TYPE "FANUC_OUTPUTS"
// stored: IsFailsafeCompliant false
   STRUCT
      SYSTEM_SIGNAL : Struct
         SYS_CMD_ENABLE : Bool;   // MACHINE HEARTBEAT (MACHINE TO GANTRY) / COMMAND ENABLE
         SYS_READY : Bool;   // SYSTEM READY
         SYS_PRG_RUNNING : Bool;   // MACHINE EMERGENCY STOP OK (MACHINE TO GANTRY) / PROGRAM RUNNING
         SYS_PRG_PAUSED : Bool;   // MACHINE SAFETY GATES OK (LOCKED)(MACHINE TO GANTRY) / PROGRAM PAUSED
         SYS_MOTION_HELD : Bool;   // MACHINE IN MANUAL MODE (MACHINE TO GANTRY) / MOTION HELD
         SYS_FAULT : Bool;   // MACHINE IN AUTO MODE(MACHINE TO GANTRY) / FAULT
         SYS_TP_ENABLED : Bool;   // MACHINE AUTO CYCLE RUNNING (MACHINE TO GANTRY) / TP ENABLED
         SYS_HOLD : Bool;   // MACHINE IS IN WARMUP CYCLE (MACHINE TO GANTRY) / ROBOT HOLD
         SPARE_1_0 : Byte;   // MACHINE IN RUN OUT MODE (MACHINE TO GANTRY)
         SPARE_2_0 : Byte;   // MACHINE PART DEMAND SOON (MACHINE TO GANTRY)
         SPARE_3_0 : Byte;
      END_STRUCT;
      GENERAL_SIGNAL : Struct
         STYLE_INIT_ACK : Bool;   // GANTRY HEARTBEAT (GANTRY TO MACHINE) / ACKNOWLEDGE INITIATE STYLE
         IN_CYCLE : Bool;   // IN CYCLE
         REQ_TO_CONT : Bool;   // GANTRY EMERGENCY STOP OK (GANTRY TO MACHINE) / REQUEST TO CONTINUE
         DRY_CYCLE : Bool;   // DRY CYCLE MODE
         RBT_100_SPD : Bool;   // GANTRY IN MANUAL MODE (GANTRY TO MACHINE) / ROBOT 100% SPEED
         RBT_HEARTBEAT : Bool;   // GANTRY IN AUTO MODE (GANTRY TO MACHINE) / ROBOT HEARTBEAT SIGNAL
         "OP_PANEL_E-STOP" : Bool;   // GANTRY IN AUTO CYCLE RUNNING (GANTRY TO MACHINE) / OPERATOR PANEL E-STOP
         "TEACH_PENDANT_E-STOP" : Bool;   // GANTRY OVERHEAD DOOR CLOSED & LOCKED (GANTRY TO MACHINE) / TEACH PENDANT E-STOP
         EXT_ENABLED : Bool;   // GANTRY IN RUN OUT COMPLETE(GANTRY TO MACHINE) / EXTERNAL E-STOP
         DEAD_ENABLED : Bool;   // GANTRY CLEAR OF MACHINE (GANTRY TO MACHINE) / DEADMAN E-STOP
         "I/O_SIMULATE" : Bool;   // GANTRY CLEAR OF FIXTURE (GANTRY TO MACHINE) / I/O SIMULATED
         SRV_DISC_OFF : Bool;   // SERVO DISABLED OFF
         SRV_BATT_ALARM : Bool;   // LOW BATTERY ALARM ON SERVO
         TASK_OK : Bool;   // TASK OK
         STEP_MODE_ON : Bool;   // STEP MODE STATUS
         AUTO_MODE_ON : Bool;   // SELECTOR SWITCH IS SET TO AUTO
         T1_MODE_ON : Bool;   // SELECTOR SWITCH IS SET TO T1
         T2_MODE_ON : Bool;   // SELECTOR SWITCH IS SET TO T2
         FENCE_OPEN : Bool;   // FENCE IS OPEN
         INTERLOCK : Bool;   // ROBOT IN INTERLOCK
         ROUT_ACTIVE : Bool;   // ROUTER ACTIVE BIT
         FAULT_RSP_ACK : Bool;   // HMI OPTION FAULT RESPONSE
         DCS_SIGN_MATCH : Bool;   // DCS SIGNATURE MATCH
         REQ_DEC_CODE : Bool;   // REQUEST DECITION
         FLT_TASK_STOPPED : Bool;   // ROBOT TASK STOPPED
         FLT_COLLISION : Bool;   // ROBOT COLLITION FAULT
         FLT_BAD_PLC_INPUT : Bool;   // BAD PLC INPUT
         FLT_GRIP_LOW_PRS : Bool;   // ROBOT GRIPPER PRESSURE LOW
         FLT_BAD_OPTN : Bool;   // BAD PLC FAULT RESPONSE
         RECOV_AT_MAIN : Bool;   // RECOVERY POINTER TO MAIN
         FLT_USER_BIT_8 : Bool;   // USER DEFINABLE FAULT BIT
         SPARE_7_7 : Bool;
         SPARE_8_0 : Byte;
         SPARE_9_0 : Byte;
      END_STRUCT;
      PROGRAM : Struct
         STYLE_PROGRAM_ACK : Byte;   // GANTRY HEARTBEAT (GANTRY TO MACHINE) / SELECT STYLE PROGRAM ACKNOWLEDGE
         DEC_CODE_ACK : Byte;   // SELECT DECITION CODE ACKNOWLEDGE
         PART_TYPE_ACK : Byte;   // GANTRY EMERGENCY STOP OK (GANTRY TO MACHINE) / PART TYPE ACKNOWLEDGE
         SPARE_13_0 : Byte;   // GANTRY EMERGENCY STOP OK (GANTRY TO MACHINE)
      END_STRUCT;
      GRIPPERS : Struct
         T1_GRIPPER_A_OPEN_REQ : Bool;   // ROBOT TOOL 1 GRIPPER A OPEN REQUEST
         T1_GRIPPER_A_CLOSE_REQ : Bool;   // ROBOT TOOL 1 GRIPPER A CLOSE REQUEST
         SPARE_14_2 : Bool;
         SPARE_14_3 : Bool;
         T1_GRIPPER_A_OPEN : Bool;   // ROBOT TOOL 1 GRIPPER A OPEN
         T1_GRIPPER_A_CLOSED : Bool;   // ROBOT TOOL 1 GRIPPER A CLOSED
         SPARE_14_6 : Bool;
         SPARE_14_7 : Bool;
         T1_GRIPPER_B_OPEN_REQ : Bool;   // ROBOT TOOL 1 GRIPPER B OPEN REQUEST
         T1_GRIPPER_B_CLOSE_REQ : Bool;   // ROBOT TOOL 1 GRIPPER B CLOSE REQUEST
         SPARE_15_2 : Bool;
         SPARE_15_3 : Bool;
         T1_GRIPPER_B_OPEN : Bool;   // ROBOT TOOL 1 GRIPPER B OPEN
         T1_GRIPPER_B_CLOSED : Bool;   // ROBOT TOOL 1 GRIPPER B CLOSED
         SPARE_15_6 : Bool;
         SPARE_15_7 : Bool;
         T1_GRIPPER_C_OPEN_REQ : Bool;   // ROBOT TOOL 1 GRIPPER C OPEN REQUEST
         T1_GRIPPER_C_CLOSE_REQ : Bool;   // ROBOT TOOL 1 GRIPPER C CLOSE REQUEST
         SPARE_16_2 : Bool;
         SPARE_16_3 : Bool;
         T1_GRIPPER_C_OPEN : Bool;   // ROBOT TOOL 1 GRIPPER C OPEN
         T1_GRIPPER_C_CLOSED : Bool;   // ROBOT TOOL 1 GRIPPER C CLOSED
         SPARE_16_6 : Bool;
         SPARE_16_7 : Bool;
         T1_GRIPPER_D_OPEN_REQ : Bool;   // ROBOT TOOL 1 GRIPPER D OPEN REQUEST
         T1_GRIPPER_D_CLOSE_REQ : Bool;   // ROBOT TOOL 1 GRIPPER D CLOSE REQUEST
         SPARE_17_2 : Bool;
         SPARE_17_3 : Bool;
         T1_GRIPPER_D_OPEN : Bool;   // ROBOT TOOL 1 GRIPPER D OPEN
         T1_GRIPPER_D_CLOSED : Bool;   // ROBOT TOOL 1 GRIPPER D CLOSED
         SPARE_17_6 : Bool;
         SPARE_17_7 : Bool;
         T1_GRIPPER_E_OPEN_REQ : Bool;   // ROBOT TOOL 1 GRIPPER E OPEN REQUEST
         T1_GRIPPER_E_CLOSE_REQ : Bool;   // ROBOT TOOL 1 GRIPPER E CLOSE REQUEST
         SPARE_18_2 : Bool;
         SPARE_18_3 : Bool;
         T1_GRIPPER_E_OPEN : Bool;   // ROBOT TOOL 1 GRIPPER E OPEN
         T1_GRIPPER_E_CLOSED : Bool;   // ROBOT TOOL 1 GRIPPER E CLOSED
         SPARE_18_6 : Bool;
         SPARE_18_7 : Bool;
         T2_GRIPPER_A_OPEN_REQ : Bool;   // ROBOT TOOL 2 GRIPPER A OPEN REQUEST
         T2_GRIPPER_A_CLOSE_REQ : Bool;   // ROBOT TOOL 2 GRIPPER A CLOSE REQUEST
         SPARE_19_2 : Bool;
         SPARE_19_3 : Bool;
         T2_GRIPPER_A_OPEN : Bool;   // ROBOT TOOL 2 GRIPPER A OPEN
         T2_GRIPPER_A_CLOSED : Bool;   // ROBOT TOOL 2 GRIPPER A CLOSED
         SPARE_19_6 : Bool;
         SPARE_19_7 : Bool;
         T2_GRIPPER_B_OPEN_REQ : Bool;   // ROBOT TOOL 2 GRIPPER B OPEN REQUEST
         T2_GRIPPER_B_CLOSE_REQ : Bool;   // ROBOT TOOL 2 GRIPPER B CLOSE REQUEST
         SPARE_20_2 : Bool;
         SPARE_20_3 : Bool;
         T2_GRIPPER_B_OPEN : Bool;   // ROBOT TOOL 2 GRIPPER B OPEN
         T2_GRIPPER_B_CLOSED : Bool;   // ROBOT TOOL 2 GRIPPER B CLOSED
         SPARE_20_6 : Bool;
         SPARE_20_7 : Bool;
         T2_GRIPPER_C_OPEN_REQ : Bool;   // ROBOT TOOL 2 GRIPPER C OPEN REQUEST
         T2_GRIPPER_C_CLOSE_REQ : Bool;   // ROBOT TOOL 2 GRIPPER C CLOSE REQUEST
         SPARE_21_2 : Bool;
         SPARE_21_3 : Bool;
         T2_GRIPPER_C_OPEN : Bool;   // ROBOT TOOL 2 GRIPPER C OPEN
         T2_GRIPPER_C_CLOSED : Bool;   // ROBOT TOOL 2 GRIPPER C CLOSED
         SPARE_21_6 : Bool;
         SPARE_21_7 : Bool;
         T2_GRIPPER_D_OPEN_REQ : Bool;   // ROBOT TOOL 2 GRIPPER D OPEN REQUEST
         T2_GRIPPER_D_CLOSE_REQ : Bool;   // ROBOT TOOL 2 GRIPPER D CLOSE REQUEST
         SPARE_22_2 : Bool;
         SPARE_22_3 : Bool;
         T2_GRIPPER_D_OPEN : Bool;   // ROBOT TOOL 2 GRIPPER D OPEN
         T2_GRIPPER_D_CLOSED : Bool;   // ROBOT TOOL 2 GRIPPER D CLOSED
         SPARE_22_6 : Bool;
         SPARE_22_7 : Bool;
         T2_GRIPPER_E_OPEN_REQ : Bool;   // ROBOT TOOL 2 GRIPPER E OPEN REQUEST
         T2_GRIPPER_E_CLOSE_REQ : Bool;   // ROBOT TOOL 2 GRIPPER E CLOSE REQUEST
         SPARE_23_2 : Bool;
         SPARE_23_3 : Bool;
         T2_GRIPPER_E_OPEN : Bool;   // ROBOT TOOL 2 GRIPPER E OPEN
         T2_GRIPPER_E_CLOSED : Bool;   // ROBOT TOOL 2 GRIPPER E CLOSED
         SPARE_23_6 : Bool;
         SPARE_23_7 : Bool;
         T1_ALL_GRIPS_OPEN_REQ : Bool;   // ROBOT TOOL 1 OPEN ALL GRIPPERS REQUEST
         T1_ALL_GRIPS_CLOSE_REQ : Bool;   // ROBOT TOOL 1 CLOSE ALL GRIPPERS REQUEST
         T1_ALL_GRIPPERS_OPEN : Bool;   // ROBOT TOOL 1 ALL GRIPPERS OPEN
         T1_ALL_GRIPPERS_CLOSED : Bool;   // ROBOT TOOL 1 ALL GRIPPERS CLOSED
         SPARE_24_4 : Bool;
         SPARE_24_5 : Bool;
         SPARE_24_6 : Bool;
         SPARE_24_7 : Bool;
         T2_ALL_GRIPS_OPEN_REQ : Bool;   // ROBOT TOOL 2 CLOSE ALL GRIPPERS REQUEST
         T2_ALL_GRIPS_CLOSE_REQ : Bool;   // ROBOT TOOL 2 CLOSE ALL GRIPPERS REQUEST
         T2_ALL_GRIPPERS_OPEN : Bool;   // ROBOT TOOL 2 ALL GRIPPERS OPEN
         T2_ALL_GRIPPERS_CLOSED : Bool;   // ROBOT TOOL 2 ALL GRIPPERS CLOSED
         SPARE_25_4 : Bool;
         SPARE_25_5 : Bool;
         SPARE_25_6 : Bool;
         SPARE_25_7 : Bool;
         SPARE_26_0 : Byte;
         FAULT_NUMBER : Byte;   // FAULT RESPONSE
      END_STRUCT;
      CLEARS : Struct
         CLEAR_U_1_ACK : Bool;   // GANTRY HEARTBEAT (GANTRY TO MACHINE) / ROBOT OUT OF UNIT 1
         CLEAR_U_2_ACK : Bool;   // ROBOT OUT OF UNIT 2
         CLEAR_U_3_ACK : Bool;   // GANTRY EMERGENCY STOP OK (GANTRY TO MACHINE) / ROBOT OUT OF UNIT 3
         CLEAR_U_4_ACK : Bool;   // ROBOT OUT OF UNIT 4
         CLEAR_U_5_ACK : Bool;   // GANTRY IN MANUAL MODE (GANTRY TO MACHINE) / ROBOT OUT OF UNIT 5
         CLEAR_U_6_ACK : Bool;   // GANTRY IN AUTO MODE (GANTRY TO MACHINE) / ROBOT OUT OF UNIT 6
         CLEAR_U_7_ACK : Bool;   // GANTRY IN AUTO CYCLE RUNNING (GANTRY TO MACHINE) / ROBOT OUT OF UNIT 7
         CLEAR_U_8_ACK : Bool;   // GANTRY OVERHEAD DOOR CLOSED & LOCKED (GANTRY TO MACHINE) / ROBOT OUT OF UNIT 8
         CLEAR_U_9_ACK : Bool;   // GANTRY IN RUN OUT COMPLETE(GANTRY TO MACHINE) / ROBOT OUT OF UNIT 9
         CLEAR_U_10_ACK : Bool;   // GANTRY CLEAR OF MACHINE (GANTRY TO MACHINE) / ROBOT OUT OF UNIT 10
         SPARE_29_2 : Bool;   // GANTRY CLEAR OF FIXTURE (GANTRY TO MACHINE)
         SPARE_29_3 : Bool;
         SPARE_29_4 : Bool;
         SPARE_29_5 : Bool;   // GANTRY PART TYPE CHANGE REQUESTED (GANTRY TO MACHINE)
         SPARE_29_6 : Bool;   // GANTRY REQUEST MACHINE TO RUN WITH LOADED PARTS (GANTRY TO MACHINE)
         SPARE_29_7 : Bool;   // GANTRY RUN OUT REQUESTED (GANTRY TO MACHINE)
         SPARE_30_0 : Byte;
         SPARE_31_0 : Byte;
      END_STRUCT;
      TASKS : Struct
         TSK_COMPLETED_1 : Bool;   // GANTRY HEARTBEAT (GANTRY TO MACHINE) / ROBOT TASK 1 COMPLETED
         TSK_COMPLETED_2 : Bool;   // ROBOT TASK 2 COMPLETED
         TSK_COMPLETED_3 : Bool;   // GANTRY EMERGENCY STOP OK (GANTRY TO MACHINE) / ROBOT TASK 3 COMPLETED
         TSK_COMPLETED_4 : Bool;   // ROBOT TASK 4 COMPLETED
         TSK_COMPLETED_5 : Bool;   // GANTRY IN MANUAL MODE (GANTRY TO MACHINE) / ROBOT TASK 5 COMPLETED
         TSK_COMPLETED_6 : Bool;   // GANTRY IN AUTO MODE (GANTRY TO MACHINE) / ROBOT TASK 6 COMPLETED
         TSK_COMPLETED_7 : Bool;   // GANTRY IN AUTO CYCLE RUNNING (GANTRY TO MACHINE) / ROBOT TASK 7 COMPLETED
         TSK_COMPLETED_8 : Bool;   // GANTRY OVERHEAD DOOR CLOSED & LOCKED (GANTRY TO MACHINE) / ROBOT TASK 8 COMPLETED
         SPARE_33_0 : Byte;   // GANTRY IN RUN OUT COMPLETE(GANTRY TO MACHINE) / ROBOT TASK 9 COMPLETED
         SPARE_34_0 : Byte;   // GANTRY CLEAR OF MACHINE (GANTRY TO MACHINE) / ROBOT TASK 10 COMPLETED
         SPARE_35_0 : Byte;   // GANTRY CLEAR OF FIXTURE (GANTRY TO MACHINE)
         SPARE_36_0 : Byte;
         SPARE_37_0 : Byte;
         SPARE_38_0 : Byte;
         SPARE_39_0 : Byte;
      END_STRUCT;
      POSITIONS : Struct
         HOME : Bool;   // GANTRY HEARTBEAT (GANTRY TO MACHINE) / ROBOT AT HOME POSITION
         MAINT : Bool;   // ROBOT AT MAINTENANCE POSITION
         REPAIR : Bool;   // GANTRY EMERGENCY STOP OK (GANTRY TO MACHINE) / ROBOT AT REPAIRED POSITION
         ALIGN : Bool;   // ROBOT AT ALIGNED POSITION
         SHIP : Bool;   // GANTRY IN MANUAL MODE (GANTRY TO MACHINE) / ROBOT AT SHIPPED POSITION
         SPARE_38_5 : Bool;   // GANTRY IN AUTO MODE (GANTRY TO MACHINE)
         SPARE_38_6 : Bool;   // GANTRY IN AUTO CYCLE RUNNING (GANTRY TO MACHINE)
         SPARE_38_7 : Bool;   // GANTRY OVERHEAD DOOR CLOSED & LOCKED (GANTRY TO MACHINE)
         UNIT_1 : Bool;   // GANTRY OVERHEAD DOOR CLOSED & LOCKED (GANTRY TO MACHINE) / ROBOT AT POUNCE POSITION UNIT 1
         UNIT_2 : Bool;   // GANTRY OVERHEAD DOOR CLOSED & LOCKED (GANTRY TO MACHINE) / ROBOT AT POUNCE POSITION UNIT 2
         UNIT_3 : Bool;   // GANTRY OVERHEAD DOOR CLOSED & LOCKED (GANTRY TO MACHINE) / ROBOT AT POUNCE POSITION UNIT 3
         UNIT_4 : Bool;   // GANTRY OVERHEAD DOOR CLOSED & LOCKED (GANTRY TO MACHINE) / ROBOT AT POUNCE POSITION UNIT 4
         UNIT_5 : Bool;   // GANTRY OVERHEAD DOOR CLOSED & LOCKED (GANTRY TO MACHINE) / ROBOT AT POUNCE POSITION UNIT 5
         UNIT_6 : Bool;   // GANTRY IN RUN OUT COMPLETE(GANTRY TO MACHINE) / ROBOT AT POUNCE POSITION UNIT 6
         UNIT_7 : Bool;   // GANTRY IN RUN OUT COMPLETE(GANTRY TO MACHINE) / ROBOT AT POUNCE POSITION UNIT 7
         UNIT_8 : Bool;   // GANTRY IN RUN OUT COMPLETE(GANTRY TO MACHINE) / ROBOT AT POUNCE POSITION UNIT 8
         SPARE_42_0 : Byte;   // GANTRY CLEAR OF MACHINE (GANTRY TO MACHINE)
         SPARE_43_0 : Byte;   // GANTRY CLEAR OF FIXTURE (GANTRY TO MACHINE)
         SPARE_44_0 : Byte;
         SPARE_45_0 : Byte;
      END_STRUCT;
      SPARES : Array[46..63] of Byte;
   END_STRUCT;
END_TYPE

TYPE "KUKA_INPUTS"
// stored: IsFailsafeCompliant false
   STRUCT
      SYSTEM_SIGNAL : Struct
         PROGRAM_NUMBER : Byte;   // MACHINE HEARTBEAT (MACHINE TO GANTRY) / PROGRAM NUMBER
         SRB : Bool;   // SRB
         ANTEIN : Bool;   // MACHINE EMERGENCY STOP OK (MACHINE TO GANTRY) / ANTEIN
         SPARE_65_2 : Bool;   // MACHINE SAFETY GATES OK (LOCKED)(MACHINE TO GANTRY)
         SPARE_65_3 : Bool;   // MACHINE IN MANUAL MODE (MACHINE TO GANTRY)
         SPARE_65_4 : Bool;   // MACHINE IN AUTO MODE(MACHINE TO GANTRY)
         SPARE_65_5 : Bool;   // MACHINE AUTO CYCLE RUNNING (MACHINE TO GANTRY)
         SPARE_65_6 : Bool;   // MACHINE IS IN WARMUP CYCLE (MACHINE TO GANTRY)
         SPARE_65_7 : Bool;
         SPARE_66_0 : Byte;   // MACHINE PART DEMAND SOON (MACHINE TO GANTRY)
         SPARE_67_0 : Byte;
      END_STRUCT;
      GENERAL_SIGNAL : Struct
         STYLE_INIT : Bool;   // GANTRY HEARTBEAT (GANTRY TO MACHINE) / INITIATE STYLE PROGRAM
         READ_DEC_CODE : Bool;   // READ DECISION CODE
         OK_CONTINUE : Bool;   // GANTRY EMERGENCY STOP OK (GANTRY TO MACHINE) / OK TO CONTINUE
         ENTER_REQUEST : Bool;   // ENTER CELL REQUEST
         DRY_CYCLE : Bool;   // GANTRY IN MANUAL MODE (GANTRY TO MACHINE) / DRY CYCLE
         RECOVER_REQ : Bool;   // GANTRY IN AUTO MODE (GANTRY TO MACHINE) / RECOVERY REQUEST
         SPARE_68_6 : Bool;   // GANTRY IN AUTO CYCLE RUNNING (GANTRY TO MACHINE)
         SPARE_68_7 : Bool;   // GANTRY OVERHEAD DOOR CLOSED & LOCKED (GANTRY TO MACHINE)
         IMMEDIATE_STOP_AUX : Bool;   // IMMEDIATE STOP AUXILIAR
         STOP_END_OF_CYCLE : Bool;   // STOP END OF CYCLE
         RUNOUT_REQUEST : Bool;   // RUNOUT REQUEST
         SPARE_69_3 : Bool;
         SPARE_69_4 : Bool;
         SPARE_69_5 : Bool;
         SPARE_69_6 : Bool;
         SPARE_69_7 : Bool;
         BRAKE_TEST_EXT_REQ : Bool;   // BRAKE TEST EXTERNAL REQUEST
         MASTER_TEST_EXT_REQ : Bool;   // MASTER TEST EXTERNAL REQUEST
         SPARE_70_2 : Bool;
         HOME_INTERRUPTION : Bool;   // HOME INTERRUPTION
         SPARE_70_4 : Bool;
         SPARE_70_5 : Bool;
         SPARE_70_6 : Bool;
         SPARE_70_7 : Bool;
         SPARE_71_0 : Byte;   // GANTRY CLEAR OF FIXTURE (GANTRY TO MACHINE)
         SPARE_72_0 : Byte;
         SPARE_73_0 : Byte;
      END_STRUCT;
      PROGRAM : Struct
         STYLE_PROGRAM : Byte;   // GANTRY HEARTBEAT (GANTRY TO MACHINE) / GROUP INPUT INDICATING STYLE NUMBER PROGRAM
         DEC_CODE : Byte;   // SPECIFIC OPERATING WITHIN A STYLE
         PART_TYPE : Byte;   // GANTRY EMERGENCY STOP OK (GANTRY TO MACHINE) / PART TYPE SELECTED
         SPARE_77_0 : Byte;   // GANTRY EMERGENCY STOP OK (GANTRY TO MACHINE)
      END_STRUCT;
      GRIPPERS : Struct
         T1_GRIPPER_A_OPEN_REQ : Bool;   // ROBOT TOOL 1 GRIPPER A OPEN REQUEST
         T1_GRIPPER_A_CLOSE_REQ : Bool;   // ROBOT TOOL 1 GRIPPER A CLOSE REQUEST
         SPARE_78_2 : Bool;
         SPARE_78_3 : Bool;
         T1_GRIPPER_A_OPEN : Bool;   // ROBOT TOOL 1 GRIPPER A OPEN
         T1_GRIPPER_A_CLOSED : Bool;   // ROBOT TOOL 1 GRIPPER A CLOSED
         SPARE_78_6 : Bool;
         SPARE_78_7 : Bool;
         T1_GRIPPER_B_OPEN_REQ : Bool;   // ROBOT TOOL 1 GRIPPER B OPEN REQUEST
         T1_GRIPPER_B_CLOSE_REQ : Bool;   // ROBOT TOOL 1 GRIPPER B CLOSE REQUEST
         SPARE_79_2 : Bool;
         SPARE_79_3 : Bool;
         T1_GRIPPER_B_OPEN : Bool;   // ROBOT TOOL 1 GRIPPER B OPEN
         T1_GRIPPER_B_CLOSED : Bool;   // ROBOT TOOL 1 GRIPPER B CLOSED
         SPARE_79_6 : Bool;
         SPARE_79_7 : Bool;
         T1_GRIPPER_C_OPEN_REQ : Bool;   // ROBOT TOOL 1 GRIPPER C OPEN REQUEST
         T1_GRIPPER_C_CLOSE_REQ : Bool;   // ROBOT TOOL 1 GRIPPER C CLOSE REQUEST
         SPARE_80_2 : Bool;
         SPARE_80_3 : Bool;
         T1_GRIPPER_C_OPEN : Bool;   // ROBOT TOOL 1 GRIPPER C OPEN
         T1_GRIPPER_C_CLOSED : Bool;   // ROBOT TOOL 1 GRIPPER C CLOSED
         SPARE_80_6 : Bool;
         SPARE_80_7 : Bool;
         T1_GRIPPER_D_OPEN_REQ : Bool;   // ROBOT TOOL 1 GRIPPER D OPEN REQUEST
         T1_GRIPPER_D_CLOSE_REQ : Bool;   // ROBOT TOOL 1 GRIPPER D CLOSE REQUEST
         SPARE_81_2 : Bool;
         SPARE_81_3 : Bool;
         T1_GRIPPER_D_OPEN : Bool;   // ROBOT TOOL 1 GRIPPER D OPEN
         T1_GRIPPER_D_CLOSED : Bool;   // ROBOT TOOL 1 GRIPPER D CLOSED
         SPARE_81_6 : Bool;
         SPARE_81_7 : Bool;
         T1_GRIPPER_E_OPEN_REQ : Bool;   // ROBOT TOOL 1 GRIPPER E OPEN REQUEST
         T1_GRIPPER_E_CLOSE_REQ : Bool;   // ROBOT TOOL 1 GRIPPER E CLOSE REQUEST
         SPARE_82_2 : Bool;
         SPARE_82_3 : Bool;
         T1_GRIPPER_E_OPEN : Bool;   // ROBOT TOOL 1 GRIPPER E OPEN
         T1_GRIPPER_E_CLOSED : Bool;   // ROBOT TOOL 1 GRIPPER E CLOSED
         SPARE_82_6 : Bool;
         SPARE_82_7 : Bool;
         T2_GRIPPER_A_OPEN_REQ : Bool;   // ROBOT TOOL 2 GRIPPER A OPEN REQUEST
         T2_GRIPPER_A_CLOSE_REQ : Bool;   // ROBOT TOOL 2 GRIPPER A CLOSE REQUEST
         SPARE_83_2 : Bool;
         SPARE_83_3 : Bool;
         T2_GRIPPER_A_OPEN : Bool;   // ROBOT TOOL 2 GRIPPER A OPEN
         T2_GRIPPER_A_CLOSED : Bool;   // ROBOT TOOL 2 GRIPPER A CLOSED
         SPARE_83_6 : Bool;
         SPARE_83_7 : Bool;
         T2_GRIPPER_B_OPEN_REQ : Bool;   // ROBOT TOOL 2 GRIPPER B OPEN REQUEST
         T2_GRIPPER_B_CLOSE_REQ : Bool;   // ROBOT TOOL 2 GRIPPER B CLOSE REQUEST
         SPARE_84_2 : Bool;
         SPARE_84_3 : Bool;
         T2_GRIPPER_B_OPEN : Bool;   // ROBOT TOOL 2 GRIPPER B OPEN
         T2_GRIPPER_B_CLOSED : Bool;   // ROBOT TOOL 2 GRIPPER B CLOSED
         SPARE_84_6 : Bool;
         SPARE_84_7 : Bool;
         T2_GRIPPER_C_OPEN_REQ : Bool;   // ROBOT TOOL 2 GRIPPER C OPEN REQUEST
         T2_GRIPPER_C_CLOSE_REQ : Bool;   // ROBOT TOOL 2 GRIPPER C CLOSE REQUEST
         SPARE_85_2 : Bool;
         SPARE_85_3 : Bool;
         T2_GRIPPER_C_OPEN : Bool;   // ROBOT TOOL 2 GRIPPER C OPEN
         T2_GRIPPER_C_CLOSED : Bool;   // ROBOT TOOL 2 GRIPPER C CLOSED
         SPARE_85_6 : Bool;
         SPARE_85_7 : Bool;
         T2_GRIPPER_D_OPEN_REQ : Bool;   // ROBOT TOOL 2 GRIPPER D OPEN REQUEST
         T2_GRIPPER_D_CLOSE_REQ : Bool;   // ROBOT TOOL 2 GRIPPER D CLOSE REQUEST
         SPARE_86_2 : Bool;
         SPARE_86_3 : Bool;
         T2_GRIPPER_D_OPEN : Bool;   // ROBOT TOOL 2 GRIPPER D OPEN
         T2_GRIPPER_D_CLOSED : Bool;   // ROBOT TOOL 2 GRIPPER D CLOSED
         SPARE_86_6 : Bool;
         SPARE_86_7 : Bool;
         T2_GRIPPER_E_OPEN_REQ : Bool;   // ROBOT TOOL 2 GRIPPER E OPEN REQUEST
         T2_GRIPPER_E_CLOSE_REQ : Bool;   // ROBOT TOOL 2 GRIPPER E CLOSE REQUEST
         SPARE_87_2 : Bool;
         SPARE_87_3 : Bool;
         T2_GRIPPER_E_OPEN : Bool;   // ROBOT TOOL 2 GRIPPER E OPEN
         T2_GRIPPER_E_CLOSED : Bool;   // ROBOT TOOL 2 GRIPPER E CLOSED
         SPARE_87_6 : Bool;
         SPARE_87_7 : Bool;
         T1_ALL_GRIPS_OPEN_REQ : Bool;   // ROBOT TOOL 1 OPEN ALL GRIPPERS REQUEST
         T1_ALL_GRIPS_CLOSE_REQ : Bool;   // ROBOT TOOL 1 CLOSE ALL GRIPPERS REQUEST
         T1_ALL_GRIPPERS_OPEN : Bool;   // ROBOT TOOL 1 ALL GRIPPERS OPEN
         T1_ALL_GRIPPERS_CLOSED : Bool;   // ROBOT TOOL 1 ALL GRIPPERS CLOSED
         SPARE_88_4 : Bool;
         SPARE_88_5 : Bool;
         SPARE_88_6 : Bool;
         SPARE_88_7 : Bool;
         T2_ALL_GRIPS_OPEN_REQ : Bool;   // ROBOT TOOL 2 CLOSE ALL GRIPPERS REQUEST
         T2_ALL_GRIPS_CLOSE_REQ : Bool;   // ROBOT TOOL 2 CLOSE ALL GRIPPERS REQUEST
         T2_ALL_GRIPPERS_OPEN : Bool;   // ROBOT TOOL 2 ALL GRIPPERS OPEN
         T2_ALL_GRIPPERS_CLOSED : Bool;   // ROBOT TOOL 2 ALL GRIPPERS CLOSED
         SPARE_89_4 : Bool;
         SPARE_89_5 : Bool;
         SPARE_89_6 : Bool;
         SPARE_89_7 : Bool;
         SPARE_90_0 : Byte;
         FAULT_NUMBER : Byte;   // FAULT RESPONSE
      END_STRUCT;
      CLEARS : Struct
         CLEAR_U_1 : Bool;   // GANTRY HEARTBEAT (GANTRY TO MACHINE) / CLEAR TO GET IN UNIT 1
         CLEAR_U_2 : Bool;   // CLEAR TO GET IN UNIT 2
         CLEAR_U_3 : Bool;   // GANTRY EMERGENCY STOP OK (GANTRY TO MACHINE) / CLEAR TO GET IN UNIT 3
         CLEAR_U_4 : Bool;   // CLEAR TO GET IN UNIT 4
         CLEAR_U_5 : Bool;   // GANTRY IN MANUAL MODE (GANTRY TO MACHINE) / CLEAR TO GET IN UNIT 5
         CLEAR_U_6 : Bool;   // GANTRY IN AUTO MODE (GANTRY TO MACHINE) / CLEAR TO GET IN UNIT 6
         CLEAR_U_7 : Bool;   // GANTRY IN AUTO CYCLE RUNNING (GANTRY TO MACHINE) / CLEAR TO GET IN UNIT 7
         CLEAR_U_8 : Bool;   // GANTRY OVERHEAD DOOR CLOSED & LOCKED (GANTRY TO MACHINE) / CLEAR TO GET IN UNIT 8
         CLEAR_U_9 : Bool;   // GANTRY IN RUN OUT COMPLETE(GANTRY TO MACHINE) / CLEAR TO GET IN UNIT 9
         CLEAR_U_10 : Bool;   // GANTRY CLEAR OF MACHINE (GANTRY TO MACHINE) / CLEAR TO GET IN UNIT 10
         SPARE_93_2 : Bool;   // GANTRY CLEAR OF FIXTURE (GANTRY TO MACHINE)
         SPARE_93_3 : Bool;
         SPARE_93_4 : Bool;
         SPARE_93_5 : Bool;   // GANTRY PART TYPE CHANGE REQUESTED (GANTRY TO MACHINE)
         SPARE_93_6 : Bool;   // GANTRY REQUEST MACHINE TO RUN WITH LOADED PARTS (GANTRY TO MACHINE)
         SPARE_93_7 : Bool;   // GANTRY RUN OUT REQUESTED (GANTRY TO MACHINE)
         SPARE_94_0 : Byte;
         SPARE_95_0 : Byte;
      END_STRUCT;
      TASKS : Struct
         COMPLETE_TSK_1 : Bool;   // GANTRY HEARTBEAT (GANTRY TO MACHINE) / ROBOT COMPLETE TASK 1
         COMPLETE_TSK_2 : Bool;   // ROBOT COMPLETE TASK 2
         COMPLETE_TSK_3 : Bool;   // GANTRY EMERGENCY STOP OK (GANTRY TO MACHINE) / ROBOT COMPLETE TASK 3
         COMPLETE_TSK_4 : Bool;   // ROBOT COMPLETE TASK 4
         COMPLETE_TSK_5 : Bool;   // GANTRY IN MANUAL MODE (GANTRY TO MACHINE) / ROBOT COMPLETE TASK 5
         COMPLETE_TSK_6 : Bool;   // GANTRY IN AUTO MODE (GANTRY TO MACHINE) / ROBOT COMPLETE TASK 6
         COMPLETE_TSK_7 : Bool;   // GANTRY IN AUTO CYCLE RUNNING (GANTRY TO MACHINE) / ROBOT COMPLETE TASK 7
         COMPLETE_TSK_8 : Bool;   // GANTRY OVERHEAD DOOR CLOSED & LOCKED (GANTRY TO MACHINE) / ROBOT COMPLETE TASK 8
         SPARE_97_0 : Byte;   // GANTRY IN RUN OUT COMPLETE(GANTRY TO MACHINE)
         SPARE_98_0 : Byte;   // GANTRY CLEAR OF MACHINE (GANTRY TO MACHINE)
         SPARE_99_0 : Byte;   // GANTRY CLEAR OF FIXTURE (GANTRY TO MACHINE)
         SPARE_100_0 : Byte;
         SPARE_101_0 : Byte;
         SPARE_102_0 : Byte;
         SPARE_103_0 : Byte;
      END_STRUCT;
      PARTS_ENABLED : Struct
         PART_A_ENABLED : Bool;   // GANTRY HEARTBEAT (GANTRY TO MACHINE) / PART A ENABLED TO WORK
         PART_B_ENABLED : Bool;   // PART B ENABLED TO WORK
         PART_C_ENABLED : Bool;   // GANTRY EMERGENCY STOP OK (GANTRY TO MACHINE) / PART C ENABLED TO WORK
         PART_D_ENABLED : Bool;   // PART D ENABLED TO WORK
         PART_E_ENABLED : Bool;   // GANTRY IN MANUAL MODE (GANTRY TO MACHINE) / PART E ENABLED TO WORK
         SPARE_104_5 : Bool;   // GANTRY IN AUTO MODE (GANTRY TO MACHINE)
         SPARE_104_6 : Bool;   // GANTRY IN AUTO CYCLE RUNNING (GANTRY TO MACHINE)
         SPARE_104_7 : Bool;   // GANTRY OVERHEAD DOOR CLOSED & LOCKED (GANTRY TO MACHINE)
         SPARE_105_0 : Byte;   // GANTRY CLEAR OF FIXTURE (GANTRY TO MACHINE)
      END_STRUCT;
      SPARES : Array[106..127] of Byte;
   END_STRUCT;
END_TYPE

TYPE "KUKA_OUTPUTS"
// stored: IsFailsafeCompliant false
   STRUCT
      SYSTEM_SIGNAL : Struct
         PROGRAM_NUMBER_MIRROR : Byte;   // MACHINE HEARTBEAT (MACHINE TO GANTRY) / PROGRAM NUMBER MIRROR A1-A8
         BEREIT : Bool;   // CONTROLLER READY A9
         RK100 : Bool;   // MACHINE EMERGENCY STOP OK (MACHINE TO GANTRY) / ENABLE START ACTUATORS A10
         RK8 : Bool;   // MACHINE IN MANUAL MODE (MACHINE TO GANTRY) / SINGLE STEP A11
         RK9 : Bool;   // MACHINE IN AUTO MODE(MACHINE TO GANTRY) / AUTOMATIC EXTERNAL A12
         RK23 : Bool;   // MACHINE AUTO CYCLE RUNNING (MACHINE TO GANTRY) / PROGRAMMING MODE A13
         LPKT : Bool;   // MACHINE IS IN WARMUP CYCLE (MACHINE TO GANTRY) / LAST POINT REACHED A14
         PFO : Bool;   // ROBOT AT ZERO POINT OF PROGRAM HOME POSITION A15
         BCO : Bool;   // ROBOT ON PATH A16
         WPROZ : Bool;   // WAIT FOR PROCESS INPUT A17
         WSLAV : Bool;   // WAIT FOR SLAVE INPUT A18
         INT_E_STOP : Bool;   // INTERNAL EMERGENCY STOP A19
         SPARE_2_3 : Bool;
         SPARE_2_4 : Bool;
         SPARE_2_5 : Bool;
         SPARE_2_6 : Bool;
         SPARE_2_7 : Bool;
         ROBOT_FOLGE_1_SELECTED : Bool;   // ROBOT FOLGE 1 SELECTED A25
         ROBOT_FOLGE_1_RUNNING : Bool;   // ROBOT FOLGE 1 RUNNING A26
         SPARE_3_2 : Bool;
         SPARE_3_3 : Bool;
         SPARE_3_4 : Bool;
         SPARE_3_5 : Bool;
         SPARE_3_6 : Bool;
         SPARE_3_7 : Bool;
      END_STRUCT;
      GENERAL_SIGNAL : Struct
         STYLE_INIT_ACK : Bool;   // GANTRY HEARTBEAT (GANTRY TO MACHINE) / ACKNOWLEDGE INITIATE STYLE
         IN_CYCLE : Bool;   // IN CYCLE
         REQ_TO_CONT : Bool;   // GANTRY EMERGENCY STOP OK (GANTRY TO MACHINE) / REQUEST TO CONTINUE
         DRY_CYCLE : Bool;   // DRY CYCLE MODE
         RBT_100_SPD : Bool;   // GANTRY IN MANUAL MODE (GANTRY TO MACHINE) / ROBOT 100% SPEED
         RBT_HEARTBEAT : Bool;   // GANTRY IN AUTO MODE (GANTRY TO MACHINE) / ROBOT HEARTBEAT SIGNAL
         "OP_PANEL_E-STOP" : Bool;   // GANTRY IN AUTO CYCLE RUNNING (GANTRY TO MACHINE) / OPERATOR PANEL E-STOP
         "TEACH_PENDANT_E-STOP" : Bool;   // GANTRY OVERHEAD DOOR CLOSED & LOCKED (GANTRY TO MACHINE) / TEACH PENDANT E-STOP
         EXT_ENABLED : Bool;   // GANTRY IN RUN OUT COMPLETE(GANTRY TO MACHINE) / EXTERNAL E-STOP
         DEAD_ENABLED : Bool;   // GANTRY CLEAR OF MACHINE (GANTRY TO MACHINE) / DEADMAN E-STOP
         "I/O_SIMULATE" : Bool;   // GANTRY CLEAR OF FIXTURE (GANTRY TO MACHINE) / I/O SIMULATED
         SRV_DISC_OFF : Bool;   // SERVO DISABLED OFF
         SRV_BATT_ALARM : Bool;   // LOW BATTERY ALARM ON SERVO
         TASK_OK : Bool;   // TASK OK
         STEP_MODE_ON : Bool;   // STEP MODE STATUS
         AUTO_MODE_ON : Bool;   // SELECTOR SWITCH IS SET TO AUTO
         T1_MODE_ON : Bool;   // SELECTOR SWITCH IS SET TO T1
         T2_MODE_ON : Bool;   // SELECTOR SWITCH IS SET TO T2
         FENCE_OPEN : Bool;   // FENCE IS OPEN
         INTERLOCK : Bool;   // ROBOT IN INTERLOCK
         ROUT_ACTIVE : Bool;   // ROUTER ACTIVE BIT
         FAULT_RSP_ACK : Bool;   // HMI OPTION FAULT RESPONSE
         DCS_SIGN_MATCH : Bool;   // DCS SIGNATURE MATCH
         REQ_DEC_CODE : Bool;   // REQUEST DECITION
         FLT_TASK_STOPPED : Bool;   // ROBOT TASK STOPPED
         FLT_COLLISION : Bool;   // ROBOT COLLITION FAULT
         FLT_BAD_PLC_INPUT : Bool;   // BAD PLC INPUT
         FLT_GRIP_LOW_PRS : Bool;   // ROBOT GRIPPER PRESSURE LOW
         FLT_BAD_OPTN : Bool;   // BAD PLC FAULT RESPONSE
         RECOV_AT_MAIN : Bool;   // RECOVERY POINTER TO MAIN
         FLT_USER_BIT_8 : Bool;   // USER DEFINABLE FAULT BIT
         SPARE_7_7 : Bool;
         SPARE_8_0 : Byte;
         SPARE_9_0 : Byte;
      END_STRUCT;
      PROGRAM : Struct
         STYLE_PROGRAM_ACK : Byte;   // GANTRY HEARTBEAT (GANTRY TO MACHINE) / STYLE PROGRAM ACKNOWLEDGE
         DEC_CODE_ACK : Byte;   // DECITION CODE ACKNOWLEDGE
         PART_TYPE_ACK : Byte;   // GANTRY EMERGENCY STOP OK (GANTRY TO MACHINE) / PART TYPE ACKNOWLEDGE
         SPARE_13_0 : Byte;   // GANTRY EMERGENCY STOP OK (GANTRY TO MACHINE)
      END_STRUCT;
      GRIPPERS : Struct
         T1_GRIPPER_A_OPEN_REQ : Bool;   // ROBOT TOOL 1 GRIPPER A OPEN REQUEST
         T1_GRIPPER_A_CLOSE_REQ : Bool;   // ROBOT TOOL 1 GRIPPER A CLOSE REQUEST
         SPARE_14_2 : Bool;
         SPARE_14_3 : Bool;
         T1_GRIPPER_A_OPENED : Bool;   // ROBOT TOOL 1 GRIPPER A OPENED
         T1_GRIPPER_A_CLOSED : Bool;   // ROBOT TOOL 1 GRIPPER A CLOSED
         SPARE_14_6 : Bool;
         SPARE_14_7 : Bool;
         T1_GRIPPER_B_OPEN_REQ : Bool;   // ROBOT TOOL 1 GRIPPER B OPEN REQUEST
         T1_GRIPPER_B_CLOSE_REQ : Bool;   // ROBOT TOOL 1 GRIPPER B CLOSE REQUEST
         SPARE_15_2 : Bool;
         SPARE_15_3 : Bool;
         T1_GRIPPER_B_OPENED : Bool;   // ROBOT TOOL 1 GRIPPER B OPENED
         T1_GRIPPER_B_CLOSED : Bool;   // ROBOT TOOL 1 GRIPPER B CLOSED
         SPARE_15_6 : Bool;
         SPARE_15_7 : Bool;
         T1_GRIPPER_C_OPEN_REQ : Bool;   // ROBOT TOOL 1 GRIPPER C OPEN REQUEST
         T1_GRIPPER_C_CLOSE_REQ : Bool;   // ROBOT TOOL 1 GRIPPER C CLOSE REQUEST
         SPARE_16_2 : Bool;
         SPARE_16_3 : Bool;
         T1_GRIPPER_C_OPENED : Bool;   // ROBOT TOOL 1 GRIPPER C OPENED
         T1_GRIPPER_C_CLOSED : Bool;   // ROBOT TOOL 1 GRIPPER C CLOSED
         SPARE_16_6 : Bool;
         SPARE_16_7 : Bool;
         T1_GRIPPER_D_OPEN_REQ : Bool;   // ROBOT TOOL 1 GRIPPER D OPEN REQUEST
         T1_GRIPPER_D_CLOSE_REQ : Bool;   // ROBOT TOOL 1 GRIPPER D CLOSE REQUEST
         SPARE_17_2 : Bool;
         SPARE_17_3 : Bool;   // ROBOT TOOL 1 GRIPPER D OPENED
         T1_GRIPPER_D_OPENED : Bool;   // ROBOT TOOL 1 GRIPPER D CLOSED
         T1_GRIPPER_D_CLOSED : Bool;
         SPARE_17_6 : Bool;
         SPARE_17_7 : Bool;   // ROBOT TOOL 1 GRIPPER E OPEN REQUEST
         T1_GRIPPER_E_OPEN_REQ : Bool;   // ROBOT TOOL 1 GRIPPER E CLOSE REQUEST
         T1_GRIPPER_E_CLOSE_REQ : Bool;
         SPARE_18_2 : Bool;
         SPARE_18_3 : Bool;   // ROBOT TOOL 1 GRIPPER E OPENED
         T1_GRIPPER_E_OPENED : Bool;   // ROBOT TOOL 1 GRIPPER E CLOSED
         T1_GRIPPER_E_CLOSED : Bool;
         SPARE_18_6 : Bool;
         SPARE_18_7 : Bool;   // ROBOT TOOL 2 GRIPPER A OPEN REQUEST
         T2_GRIPPER_A_OPEN_REQ : Bool;   // ROBOT TOOL 2 GRIPPER A CLOSE REQUEST
         T2_GRIPPER_A_CLOSE_REQ : Bool;
         SPARE_19_2 : Bool;
         SPARE_19_3 : Bool;   // ROBOT TOOL 2 GRIPPER A OPENED
         T2_GRIPPER_A_OPENED : Bool;   // ROBOT TOOL 2 GRIPPER A CLOSED
         T2_GRIPPER_A_CLOSED : Bool;
         SPARE_19_6 : Bool;
         SPARE_19_7 : Bool;   // ROBOT TOOL 2 GRIPPER B OPEN REQUEST
         T2_GRIPPER_B_OPEN_REQ : Bool;   // ROBOT TOOL 2 GRIPPER B CLOSE REQUEST
         T2_GRIPPER_B_CLOSE_REQ : Bool;
         SPARE_20_2 : Bool;
         SPARE_20_3 : Bool;   // ROBOT TOOL 2 GRIPPER B OPENED
         T2_GRIPPER_B_OPENED : Bool;   // ROBOT TOOL 2 GRIPPER B CLOSED
         T2_GRIPPER_B_CLOSED : Bool;
         SPARE_20_6 : Bool;
         SPARE_20_7 : Bool;   // ROBOT TOOL 2 GRIPPER C OPEN REQUEST
         T2_GRIPPER_C_OPEN_REQ : Bool;   // ROBOT TOOL 2 GRIPPER C CLOSE REQUEST
         T2_GRIPPER_C_CLOSE_REQ : Bool;
         SPARE_21_2 : Bool;
         SPARE_21_3 : Bool;   // ROBOT TOOL 2 GRIPPER C OPENED
         T2_GRIPPER_C_OPENED : Bool;   // ROBOT TOOL 2 GRIPPER C CLOSED
         T2_GRIPPER_C_CLOSED : Bool;
         SPARE_21_6 : Bool;
         SPARE_21_7 : Bool;   // ROBOT TOOL 2 GRIPPER D OPEN REQUEST
         T2_GRIPPER_D_OPEN_REQ : Bool;   // ROBOT TOOL 2 GRIPPER D CLOSE REQUEST
         T2_GRIPPER_D_CLOSE_REQ : Bool;
         SPARE_22_2 : Bool;
         SPARE_22_3 : Bool;   // ROBOT TOOL 2 GRIPPER D OPENED
         T2_GRIPPER_D_OPENED : Bool;   // ROBOT TOOL 2 GRIPPER D CLOSED
         T2_GRIPPER_D_CLOSED : Bool;
         SPARE_22_6 : Bool;
         SPARE_22_7 : Bool;   // ROBOT TOOL 2 GRIPPER E OPEN REQUEST
         T2_GRIPPER_E_OPEN_REQ : Bool;   // ROBOT TOOL 2 GRIPPER E CLOSE REQUEST
         T2_GRIPPER_E_CLOSE_REQ : Bool;
         SPARE_23_2 : Bool;
         SPARE_23_3 : Bool;   // ROBOT TOOL 2 GRIPPER E OPENED
         T2_GRIPPER_E_OPENED : Bool;   // ROBOT TOOL 2 GRIPPER E CLOSED
         T2_GRIPPER_E_CLOSED : Bool;
         SPARE_23_6 : Bool;
         SPARE_23_7 : Bool;
         T1_ALL_GRIPS_OPEN_REQ : Bool;   // ROBOT TOOL 1 OPEN ALL GRIPPERS REQUEST
         T1_ALL_GRIPS_CLOSE_REQ : Bool;   // ROBOT TOOL 1 CLOSE ALL GRIPPERS REQUEST
         T1_ALL_GRIPPERS_OPENED : Bool;   // ROBOT TOOL 1 ALL GRIPPERS OPENED
         T1_ALL_GRIPPERS_CLOSED : Bool;   // ROBOT TOOL 1 ALL GRIPPERS CLOSED
         SPARE_24_4 : Bool;
         SPARE_24_5 : Bool;
         SPARE_24_6 : Bool;
         SPARE_24_7 : Bool;
         T2_ALL_GRIPS_OPEN_REQ : Bool;   // ROBOT TOOL 2 CLOSE ALL GRIPPERS REQUEST
         T2_ALL_GRIPS_CLOSE_REQ : Bool;   // ROBOT TOOL 2 CLOSE ALL GRIPPERS REQUEST
         T2_ALL_GRIPPERS_OPENED : Bool;   // ROBOT TOOL 2 ALL GRIPPERS OPENED
         T2_ALL_GRIPPERS_CLOSED : Bool;   // ROBOT TOOL 2 ALL GRIPPERS CLOSED
         SPARE_25_4 : Bool;
         SPARE_25_5 : Bool;
         SPARE_25_6 : Bool;
         SPARE_25_7 : Bool;
         SPARE_26_0 : Byte;
         FAULT_NUMBER : Byte;   // FAULT RESPONSE
      END_STRUCT;
      CLEARS : Struct
         CLEAR_U_1_ACK : Bool;   // GANTRY HEARTBEAT (GANTRY TO MACHINE) / ROBOT OUT OF UNIT 1
         CLEAR_U_2_ACK : Bool;   // ROBOT OUT OF UNIT 2
         CLEAR_U_3_ACK : Bool;   // GANTRY EMERGENCY STOP OK (GANTRY TO MACHINE) / ROBOT OUT OF UNIT 3
         CLEAR_U_4_ACK : Bool;   // ROBOT OUT OF UNIT 4
         CLEAR_U_5_ACK : Bool;   // GANTRY IN MANUAL MODE (GANTRY TO MACHINE) / ROBOT OUT OF UNIT 5
         CLEAR_U_6_ACK : Bool;   // GANTRY IN AUTO MODE (GANTRY TO MACHINE) / ROBOT OUT OF UNIT 6
         CLEAR_U_7_ACK : Bool;   // GANTRY IN AUTO CYCLE RUNNING (GANTRY TO MACHINE) / ROBOT OUT OF UNIT 7
         CLEAR_U_8_ACK : Bool;   // GANTRY OVERHEAD DOOR CLOSED & LOCKED (GANTRY TO MACHINE) / ROBOT OUT OF UNIT 8
         CLEAR_U_9_ACK : Bool;   // GANTRY IN RUN OUT COMPLETE(GANTRY TO MACHINE) / ROBOT OUT OF UNIT 9
         CLEAR_U_10_ACK : Bool;   // GANTRY CLEAR OF MACHINE (GANTRY TO MACHINE) / ROBOT OUT OF UNIT 10
         SPARE_29_2 : Bool;   // GANTRY CLEAR OF FIXTURE (GANTRY TO MACHINE)
         SPARE_29_3 : Bool;
         SPARE_29_4 : Bool;
         SPARE_29_5 : Bool;   // GANTRY PART TYPE CHANGE REQUESTED (GANTRY TO MACHINE)
         SPARE_29_6 : Bool;   // GANTRY REQUEST MACHINE TO RUN WITH LOADED PARTS (GANTRY TO MACHINE)
         SPARE_29_7 : Bool;   // GANTRY RUN OUT REQUESTED (GANTRY TO MACHINE)
         SPARE_30_0 : Byte;
         SPARE_31_0 : Byte;
      END_STRUCT;
      TASKS : Struct
         TSK_COMPLETED_1 : Bool;   // GANTRY HEARTBEAT (GANTRY TO MACHINE) / ROBOT TASK 1 COMPLETED
         TSK_COMPLETED_2 : Bool;   // ROBOT TASK 2 COMPLETED
         TSK_COMPLETED_3 : Bool;   // GANTRY EMERGENCY STOP OK (GANTRY TO MACHINE) / ROBOT TASK 3 COMPLETED
         TSK_COMPLETED_4 : Bool;   // ROBOT TASK 4 COMPLETED
         TSK_COMPLETED_5 : Bool;   // GANTRY IN MANUAL MODE (GANTRY TO MACHINE) / ROBOT TASK 5 COMPLETED
         TSK_COMPLETED_6 : Bool;   // GANTRY IN AUTO MODE (GANTRY TO MACHINE) / ROBOT TASK 6 COMPLETED
         TSK_COMPLETED_7 : Bool;   // GANTRY IN AUTO CYCLE RUNNING (GANTRY TO MACHINE) / ROBOT TASK 7 COMPLETED
         TSK_COMPLETED_8 : Bool;   // GANTRY OVERHEAD DOOR CLOSED & LOCKED (GANTRY TO MACHINE) / ROBOT TASK 8 COMPLETED
         TSK_COMPLETED_9 : Byte;   // GANTRY IN RUN OUT COMPLETE(GANTRY TO MACHINE) / ROBOT TASK 9 COMPLETED
         TSK_COMPLETED_10 : Byte;   // GANTRY CLEAR OF MACHINE (GANTRY TO MACHINE) / ROBOT TASK 10 COMPLETED
         SPARE_35_0 : Byte;   // GANTRY CLEAR OF FIXTURE (GANTRY TO MACHINE)
         SPARE_36_0 : Byte;
         SPARE_37_0 : Byte;
         SPARE_38_0 : Byte;
         SPARE_39_0 : Byte;
      END_STRUCT;
      POSITIONS : Struct
         HOME : Bool;   // GANTRY HEARTBEAT (GANTRY TO MACHINE) / ROBOT AT HOME POSITION
         MAINT : Bool;   // ROBOT AT MAINTENANCE POSITION
         REPAIR : Bool;   // GANTRY EMERGENCY STOP OK (GANTRY TO MACHINE) / ROBOT AT REPAIRED POSITION
         ALIGN : Bool;   // ROBOT AT ALIGNED POSITION
         SHIP : Bool;   // GANTRY IN MANUAL MODE (GANTRY TO MACHINE) / ROBOT AT SHIPPED POSITION
         SPARE_38_5 : Bool;   // GANTRY IN AUTO MODE (GANTRY TO MACHINE)
         SPARE_38_6 : Bool;   // GANTRY IN AUTO CYCLE RUNNING (GANTRY TO MACHINE)
         SPARE_38_7 : Bool;   // GANTRY OVERHEAD DOOR CLOSED & LOCKED (GANTRY TO MACHINE)
         UNIT_1 : Bool;   // GANTRY OVERHEAD DOOR CLOSED & LOCKED (GANTRY TO MACHINE) / ROBOT AT POUNCE POSITION UNIT 1
         UNIT_2 : Bool;   // GANTRY OVERHEAD DOOR CLOSED & LOCKED (GANTRY TO MACHINE) / ROBOT AT POUNCE POSITION UNIT 2
         UNIT_3 : Bool;   // GANTRY OVERHEAD DOOR CLOSED & LOCKED (GANTRY TO MACHINE) / ROBOT AT POUNCE POSITION UNIT 3
         UNIT_4 : Bool;   // GANTRY OVERHEAD DOOR CLOSED & LOCKED (GANTRY TO MACHINE) / ROBOT AT POUNCE POSITION UNIT 4
         UNIT_5 : Bool;   // GANTRY OVERHEAD DOOR CLOSED & LOCKED (GANTRY TO MACHINE) / ROBOT AT POUNCE POSITION UNIT 5
         UNIT_6 : Bool;   // GANTRY IN RUN OUT COMPLETE(GANTRY TO MACHINE) / ROBOT AT POUNCE POSITION UNIT 6
         UNIT_7 : Bool;   // GANTRY IN RUN OUT COMPLETE(GANTRY TO MACHINE) / ROBOT AT POUNCE POSITION UNIT 7
         UNIT_8 : Bool;   // GANTRY IN RUN OUT COMPLETE(GANTRY TO MACHINE) / ROBOT AT POUNCE POSITION UNIT 8
         SPARE_42_0 : Byte;   // GANTRY CLEAR OF MACHINE (GANTRY TO MACHINE)
         SPARE_43_0 : Byte;   // GANTRY CLEAR OF FIXTURE (GANTRY TO MACHINE)
         SPARE_44_0 : Byte;
         SPARE_45_0 : Byte;
      END_STRUCT;
      SPARES : Array[46..63] of Byte;
   END_STRUCT;
END_TYPE

TYPE "LOAD_ROBOT"
// stored: IsFailsafeCompliant false
   STRUCT
      TO_FIXT : Struct
         PART_A_LOADED_FIXT1 : Bool;   // PART 1 LOADED ARM 1 / PART A LOADED FIXT 1
         PART_B_LOADED_FIXT1 : Bool;   // PART 2 LOADED ARM 1 / PART B LOADED FIXT 1
         PART_C_LOADED_FIXT1 : Bool;   // PART 3 LOADED ARM 1 / PART C LOADED FIXT 1
         PART_D_LOADED_FIXT1 : Bool;   // PART 4 LOADED ARM 1 / PART D LOADED FIXT 1
         PART_A_LOADED_FIXT2 : Bool;   // PART 1 LOADED ARM 2 / PART A LOADED FIXT 2
         PART_B_LOADED_FIXT2 : Bool;   // PART 2 LOADED ARM 2 / PART B LOADED FIXT 2
         PART_C_LOADED_FIXT2 : Bool;   // PART 3 LOADED ARM 2 / PART C LOADED FIXT 2
         PART_D_LOADED_FIXT2 : Bool;   // PART 4 LOADED ARM 2 / PART D LOADED FIXT 2
         PARTS_LOADED_FIXT1 : Bool;   // PARTS LOADED ARM 1 / PARTS LOADED FIXT 1
         PARTS_LOADED_FIXT2 : Bool;   // PARTS LOADED ARM 2 / PARTS LOADED FIXT 2
         I_PART_PRESENT_A : Bool;   // INPUT PART PRESENT A
         I_PART_PRESENT_B : Bool;   // INPUT PART PRESENT B
         I_PART_PRESENT_C : Bool;   // INPUT PART PRESENT C
         I_PART_PRESENT_D : Bool;   // INPUT PART PRESENT D
         PART_A_UNLOADED_FIXT1 : Bool;   // PART 1 UNLOADED ARM 1 / PART A UNLOADED FIXT 1
         PART_B_UNLOADED_FIXT1 : Bool;   // PART 2 UNLOADED ARM 1 / PART B UNLOADED FIXT 1
         PART_C_UNLOADED_FIXT1 : Bool;   // PART 3 UNLOADED ARM 1 / PART C UNLOADED FIXT 1
         PART_D_UNLOADED_FIXT1 : Bool;   // PART 4 UNLOADED ARM 1 / PART D UNLOADED FIXT 1
         PART_A_UNLOADED_FIXT2 : Bool;   // PART 1 UNLOADED ARM 2 / PART A UNLOADED FIXT 2
         PART_B_UNLOADED_FIXT2 : Bool;   // PART 2 UNLOADED ARM 2 / PART B UNLOADED FIXT 2
         PART_C_UNLOADED_FIXT2 : Bool;   // PART 3 UNLOADED ARM 2 / PART C UNLOADED FIXT 2
         PART_D_UNLOADED_FIXT2 : Bool;   // PART 4 UNLOADED ARM 2 / PART D UNLOADED FIXT 2
         PARTS_UNLOADED_FIXT1 : Bool;   // PARTS UNLOADED ARM 1 / PARTS UNLOADED FIXT 1
         PARTS_UNLOADED_FIXT2 : Bool;   // PARTS UNLOADED ARM 2 / PARTS UNLOADED FIXT 2
         AUX_PART_A_LOADED_FIXT1 : Bool;   // AUX PART A LOADED FIXT1
         AUX_PART_B_LOADED_FIXT1 : Bool;   // AUX PART B LOADED FIXT1
         AUX_PART_C_LOADED_FIXT1 : Bool;   // AUX PART C LOADED FIXT1
         AUX_PART_D_LOADED_FIXT1 : Bool;   // AUX PART D LOADED FIXT1
         AUX_PART_A_LOADED_FIXT2 : Bool;   // AUX PART A LOADED FIXT2
         AUX_PART_B_LOADED_FIXT2 : Bool;   // AUX PART B LOADED FIXT2
         AUX_PART_C_LOADED_FIXT2 : Bool;   // AUX PART C LOADED FIXT2
         AUX_PART_D_LOADED_FIXT2 : Bool;   // AUX PART D LOADED FIXT2
         NO_PARTS_AT_FIXT1 : Bool;   // NO PARTS AT ARM 1 / NO PARTS AT FIXT 1
         NO_PARTS_AT_FIXT2 : Bool;   // NO PARTS AT ARM 2 / NO PARTS AT FIXT 2
         PART_A_LOADED_FIXT1_P : Bool;   // PART 1 LOADED ARM 1 PULSE / PART A LOADED FIXT 1 PULSE
         PART_B_LOADED_FIXT1_P : Bool;   // PART 2 LOADED ARM 1 PULSE / PART B LOADED FIXT 1 PULSE
         PART_C_LOADED_FIXT1_P : Bool;   // PART 3 LOADED ARM 1 PULSE / PART C LOADED FIXT 1 PULSE
         PART_D_LOADED_FIXT1_P : Bool;   // PART 4 LOADED ARM 1 PULSE / PART D LOADED FIXT 1 PULSE
         PART_A_LOADED_FIXT2_P : Bool;   // PART 1 LOADED ARM 2 PULSE / PART A LOADED FIXT 2 PULSE
         PART_B_LOADED_FIXT2_P : Bool;   // PART 2 LOADED ARM 2 PULSE / PART B LOADED FIXT 2 PULSE
         PART_C_LOADED_FIXT2_P : Bool;   // PART 3 LOADED ARM 2 PULSE / PART C LOADED FIXT 2 PULSE
         PART_D_LOADED_FIXT2_P : Bool;   // PART 4 LOADED ARM 2 PULSE / PART D LOADED FIXT 2 PULSE
         PARTS_LOADED_FIXT1_P : Bool;   // PARTS LOADED ARM 1 PULSE / PARTS LOADED FIXT 1 PULSE
         PARTS_LOADED_FIXT2_P : Bool;   // PARTS LOADED ARM 2 PULSE / PARTS LOADED FIXT 2 PULSE
         ANY_PART_LOADED : Bool;   // ANY PART LOADED
         ANY_PART_UNLOADED : Bool;   // ANY PART UNLOADED
         ENABLE_LOAD_UNLOAD : Bool;   // ENABLE TO LOAD UNLOAD LOADER TO TRANSFER
         PARTS_LOADING : Bool;   // THE GANTRY IS LOADING PARTS
         PART_A_UNLOADED_FIXT1_P : Bool;   // PART 1 UNLOADED ARM 1 PULSE / PART A UNLOADED FIXT 1 PULSE
         PART_B_UNLOADED_FIXT1_P : Bool;   // PART 2 UNLOADED ARM 1 PULSE / PART B UNLOADED FIXT 1 PULSE
         PART_C_UNLOADED_FIXT1_P : Bool;   // PART 3 UNLOADED ARM 1 PULSE / PART C UNLOADED FIXT 1 PULSE
         PART_D_UNLOADED_FIXT1_P : Bool;   // PART 4 UNLOADED ARM 1 PULSE / PART D UNLOADED FIXT 1 PULSE
         PART_A_UNLOADED_FIXT2_P : Bool;   // PART 1 UNLOADED ARM 2 PULSE / PART A UNLOADED FIXT 2 PULSE
         PART_B_UNLOADED_FIXT2_P : Bool;   // PART 2 UNLOADED ARM 2 PULSE / PART B UNLOADED FIXT 2 PULSE
         PART_C_UNLOADED_FIXT2_P : Bool;   // PART 3 UNLOADED ARM 2 PULSE / PART C UNLOADED FIXT 2 PULSE
         PART_D_UNLOADED_FIXT2_P : Bool;   // PART 4 UNLOADED ARM 2 PULSE / PART D UNLOADED FIXT 2 PULSE
         PARTS_UNLOADED_FIXT1_P : Bool;   // PARTS UNLOADED ARM 1 PULSE / PARTS UNLOADED FIXT 1 PULSE
         PARTS_UNLOADED_FIXT2_P : Bool;   // PARTS UNLOADED ARM 2 PULSE / PARTS UNLOADED FIXT 2 PULSE
         PARTS_UNLOADING : Bool;   // THE GANTRY IS UNLOADING PARTS
         ACK_REJECT_PART_A_FX2 : Bool;   // ACKNOWLEDGE REJECT PART A FROM FIXTURE 2
         ACK_REJECT_PART_B_FX2 : Bool;   // ACKNOWLEDGE REJECT PART B FROM FIXTURE 2
         ACK_REJECT_PART_C_FX2 : Bool;   // ACKNOWLEDGE REJECT PART C FROM FIXTURE 2
         ACK_REJECT_PART_D_FX2 : Bool;   // ACKNOWLEDGE REJECT PART D FROM FIXTURE 2
      END_STRUCT;
      FROM_FIXT : Struct
         REQ_LOAD_PART_A_FIXT1 : Bool;   // REQUEST LOAD PART 1 ARM 1 / REQUEST LOAD PART A FIXT 1
         REQ_LOAD_PART_B_FIXT1 : Bool;   // REQUEST LOAD PART 2 ARM 1 / REQUEST LOAD PART B FIXT 1
         REQ_LOAD_PART_C_FIXT1 : Bool;   // REQUEST LOAD PART 3 ARM 1 / REQUEST LOAD PART C FIXT 1
         REQ_LOAD_PART_D_FIXT1 : Bool;   // REQUEST LOAD PART 4 ARM 1 / REQUEST LOAD PART D FIXT 1
         REQ_LOAD_PART_A_FIXT2 : Bool;   // REQUEST LOAD PART 1 ARM 2 / REQUEST LOAD PART A FIXT 2
         REQ_LOAD_PART_B_FIXT2 : Bool;   // REQUEST LOAD PART 2 ARM 2 / REQUEST LOAD PART B FIXT 2
         REQ_LOAD_PART_C_FIXT2 : Bool;   // REQUEST LOAD PART 3 ARM 2 / REQUEST LOAD PART C FIXT 2
         REQ_LOAD_PART_D_FIXT2 : Bool;   // REQUEST LOAD PART 4 ARM 2 / REQUEST LOAD PART D FIXT 2
         REQUEST_LOAD_PARTS : Bool;   // REQUEST LOAD PARTS
         REQ_UNLOAD_PART_A_FIXT1 : Bool;   // REQUEST UNLOAD PART 1 ARM 1 / REQUEST UNLOAD PART A FIXT 1
         REQ_UNLOAD_PART_B_FIXT1 : Bool;   // REQUEST UNLOAD PART 2 ARM 1 / REQUEST UNLOAD PART B FIXT 1
         REQ_UNLOAD_PART_C_FIXT1 : Bool;   // REQUEST UNLOAD PART 3 ARM 1 / REQUEST UNLOAD PART C FIXT 1
         REQ_UNLOAD_PART_D_FIXT1 : Bool;   // REQUEST UNLOAD PART 4 ARM 1 / REQUEST UNLOAD PART D FIXT 1
         REQ_UNLOAD_PART_A_FIXT2 : Bool;   // REQUEST UNLOAD PART 1 ARM 2 / REQUEST UNLOAD PART A FIXT 2
         REQ_UNLOAD_PART_B_FIXT2 : Bool;   // REQUEST UNLOAD PART 2 ARM 2 / REQUEST UNLOAD PART B FIXT 2
         REQ_UNLOAD_PART_C_FIXT2 : Bool;   // REQUEST UNLOAD PART 3 ARM 2 / REQUEST UNLOAD PART C FIXT 2
         REQ_UNLOAD_PART_D_FIXT2 : Bool;   // REQUEST UNLOAD PART 4 ARM 2 / REQUEST UNLOAD PART D FIXT 2
         REQUEST_UNLOAD_PARTS : Bool;   // REQUEST UNLOAD PARTS
         PART_ID : Byte;   // PART ID
         NEST_FIXTURE : Byte;   // NEST FIXTURE
         PART_TYPE : Byte;   // PART TYPE
         PART_TYPE_NEST_UNLD : Byte;   // PART TYPE NEST UNLOAD
         BYTE8 : Byte;
         BYTE9 : Byte;
         BYTE10 : Byte;
         MACHINE_READY_FOR_OPERAT : Bool;   // MACHINED READY FOR OPERATION
      END_STRUCT;
   END_STRUCT;
END_TYPE

TYPE "ROBOT_GRIPPER"
// stored: IsFailsafeCompliant false
   STRUCT
      CLOSED_1_I : Bool;   // CLOSED 1 INPUT
      CLOSED_2_I : Bool;   // CLOSED 2 INPUT
      OPEN_1_I : Bool;   // OPEN 1 INPUT
      OPEN_2_I : Bool;   // OPEN 2 INPUT
      GENERAL_CONDITIONS : Bool;   // GENERAL CONDITIONS
      CLOSE_CONDITIONS : Bool;   // CLOSE CONDITIONS
      OPEN_CONDITIONS : Bool;   // OPEN CONDITIONS
      GENERAL_CONDITIONS_HELP : Bool;   // GENERAL CONDITIONS HELP
      CLOSE_CONDITIONS_HELP : Bool;   // CLOSE CONDITIONS HELP
      OPEN_CONDITIONS_HELP : Bool;   // OPEN CONDITIONS HELP
      HMI_CLOSE_MAN_REQUEST : Bool;   // HMI CLOSE MANUAL REQUEST
      HMI_CLOSE_INDPNDT_MAN_REQUEST : Bool;   // HMI CLOSE INDPNDT MANUAL REQUEST
      CLOSE_MANUAL_REQUEST : Bool;   // CLOSE MANUAL REQUEST
      HMI_OPEN_MAN_REQUEST : Bool;   // HMI OPEN MANUAL REQUEST
      HMI_OPEN_INDPNDT_MAN_REQUEST : Bool;   // HMI OPEN INDPNDT MANUAL REQUEST
      OPEN_MANUAL_REQUEST : Bool;   // OPEN MANUAL REQUEST
      CLOSE_AUTO_REQUEST : Bool;   // CLOSE AUTO REQUEST / CLOSE AUTOMATIC REQUEST
      OPEN_AUTO_REQUEST : Bool;   // OPEN AUTO REQUEST / OPEN AUTOMATIC REQUEST
      CLOSE_GLOBAL_REQUEST : Bool;   // CLOSE GLOBAL REQUEST
      OPEN_GLOBAL_REQUEST : Bool;   // OPEN GLOBAL REQUEST
      CLOSE_COMMAND : Bool;   // CLOSE COMMAND
      OPEN_COMMAND : Bool;   // OPEN COMMAND
      GENERAL_COND_HELP : Bool;   // GENERAL CONDITION HELP
      SIMULTANEITY_FAULT : Bool;   // SIMULTANEITY FAULT
      TIME_EXCEEDED : Bool;   // TIME EXCEEDED
      ALARM : Bool;   // FAULT / ALARM
      PULSE_1 : Bool;   // PULSE 1
      PULSE_2 : Bool;   // PULSE 2
      PULSE_3 : Bool;   // PULSE 3
      AUX_1 : Bool;   // AUXILIARY 1 / AUX 1
      AUX_2 : Bool;   // AUXILIARY 2 / AUX 2
      AUX_3 : Bool;   // AUXILIARY 3 / AUX 3
      AUX_4 : Bool;   // AUXILIARY 4 / AUX 4
   END_STRUCT;
END_TYPE

TYPE "ROBOT_TOOL_STATUS"
// stored: IsFailsafeCompliant false
   STRUCT
      EMPTY : Bool;   // ROBOT TOOL GRIPPER EMPTY
      ANY_PART_PRESENT : Bool;   // ROBOT TOOL GRIPPER ANY PART PRESENT
      ALL_PARTS_PRESENT : Bool;   // ROBOT TOOL GRIPPER ALL PARTS PRESENT
      SPARE_0_3 : Bool;
      SPARE_0_4 : Bool;
      SPARE_0_5 : Bool;
      SPARE_0_6 : Bool;
      SPARE_0_7 : Bool;
      PART_A_PRESENT_INPUT : Bool;   // PART A PRESENT INPUT
      PART_B_PRESENT_INPUT : Bool;   // PART B PRESENT_INPUT
      PART_C_PRESENT_INPUT : Bool;   // PART C PRESENT INPUT
      PART_D_PRESENT_INPUT : Bool;   // PART D PRESENT INPUT
      PART_E_PRESENT_INPUT : Bool;   // PART E PRESENT INPUT
      SPARE_1_5 : Bool;
      SPARE_1_6 : Bool;
      SPARE_1_7 : Bool;
      DISCORDANCY_PART_A : Bool;   // DISCORDANCY PART A
      DISCORDANCY_PART_B : Bool;   // DISCORDANCY PART B
      DISCORDANCY_PART_C : Bool;   // DISCORDANCY PART C
      DISCORDANCY_PART_D : Bool;   // DISCORDANCY PART D
      DISCORDANCY_PART_E : Bool;   // DISCORDANCY PART E
      SPARE_2_5 : Bool;
      SPARE_2_6 : Bool;
      DISCORDANCY_FAULT : Bool;   // DISCORDANCY FAULT
      ANY_NEW_PART_PRESENT : Bool;   // ANY NEW PART PRESENT
      ALL_NEW_PARTS_PRESENT : Bool;   // ALL NEW PARTS PRESENT
      NEW_PART_A : Bool;
      NEW_PART_B : Bool;
      NEW_PART_C : Bool;
      NEW_PART_D : Bool;
      NEW_PART_E : Bool;
      SPARE_3_7 : Bool;
      ANY_FNSHD_PART_PRESENT_U1 : Bool;   // ANY FINISHED PART PRESENT FROM UNIT 1
      ALL_FNSHD_PART_PRESENT_U1 : Bool;   // ALL FINISHED PARTS PRESENT FROM UNIT 1
      FINISHED_FROM_U1_PA : Bool;   // PART FINISHED FROM UNIT 1 - PART "A"
      FINISHED_FROM_U1_PB : Bool;   // PART FINISHED FROM UNIT 1 - PART "B"
      FINISHED_FROM_U1_PC : Bool;   // PART FINISHED FROM UNIT 1 - PART "C"
      FINISHED_FROM_U1_PD : Bool;   // PART FINISHED FROM UNIT 1 - PART "D"
      FINISHED_FROM_U1_PE : Bool;   // PART FINISHED FROM UNIT 1 - PART "E"
      SPARE_4_7 : Bool;
      ANY_FNSHD_PART_PRESENT_U2 : Bool;   // ANY FINISHED PART PRESENT FROM UNIT 2
      ALL_FNSHD_PART_PRESENT_U2 : Bool;   // ALL FINISHED PARTS PRESENT FROM UNIT 2
      FINISHED_FROM_U2_PA : Bool;   // PART FINISHED FROM UNIT 2 - PART "A"
      FINISHED_FROM_U2_PB : Bool;   // PART FINISHED FROM UNIT 2 - PART "B"
      FINISHED_FROM_U2_PC : Bool;   // PART FINISHED FROM UNIT 2 - PART "C"
      FINISHED_FROM_U2_PD : Bool;   // PART FINISHED FROM UNIT 2 - PART "D"
      FINISHED_FROM_U2_PE : Bool;   // PART FINISHED FROM UNIT 2 - PART "E"
      SPARE_5_7 : Bool;
      SPARE_6_0 : Byte;
      SPARE_7_0 : Byte;
      SPARE_8_0 : Byte;
      SPARE_9_0 : Byte;
      ANY_PART_REJECTED_U1 : Bool;   // ANY PART REJECTED FROM UNIT 1
      ALL_PARTS_REJTD_PRESENT_U1 : Bool;   // ALL PARTS REJECTED FROM UNIT 1
      REJECTED_FROM_U1_PA : Bool;   // REJECTED FROM UNIT 1 - PART "A"
      REJECTED_FROM_U1_PB : Bool;   // REJECTED FROM UNIT 1 - PART "B"
      REJECTED_FROM_U1_PC : Bool;   // REJECTED FROM UNIT 1 - PART "C"
      REJECTED_FROM_U1_PD : Bool;   // REJECTED FROM UNIT 1 - PART "D"
      REJECTED_FROM_U1_PE : Bool;   // REJECTED FROM UNIT 1 - PART "E"
      SPARE_10_5 : Bool;
      ANY_PART_REJECTED_U2 : Bool;   // ANY PART REJECTED FROM UNIT 2
      ALL_PARTS_REJTD_PRESENT_U2 : Bool;   // ALL PARTS REJECTED FROM UNIT 2
      REJECTED_FROM_U2_PA : Bool;   // REJECTED FROM UNIT 2 - PART "A"
      REJECTED_FROM_U2_PB : Bool;   // REJECTED FROM UNIT 2 - PART "B"
      REJECTED_FROM_U2_PC : Bool;   // REJECTED FROM UNIT 2 - PART "C"
      REJECTED_FROM_U2_PD : Bool;   // REJECTED FROM UNIT 2 - PART "D"
      REJECTED_FROM_U2_PE : Bool;   // REJECTED FROM UNIT 2 - PART "E"
      SPARE_11_5 : Bool;
      SPARE_11_6 : Bool;
      SPARE_11_7 : Bool;
      SPARE_12_0 : Byte;
      SPARE_13_0 : Byte;
      ANY_QC_PART_U1_PA : Bool;   // ANY PART TO QUALITY CHECK FROM UNIT 1
      ALL_QC_PART_U1_PA : Bool;   // ALL PARTS TO QUALITY CHECK FROM UNIT 1
      QC_FROM_U1_PA : Bool;   // QUALITY CHECK FROM UNIT 1 - PART "A"
      QC_FROM_U1_PB : Bool;   // QUALITY CHECK FROM UNIT 1 - PART "B"
      QC_FROM_U1_PC : Bool;   // QUALITY CHECK FROM UNIT 1 - PART "C"
      QC_FROM_U1_PD : Bool;   // QUALITY CHECK FROM UNIT 1 - PART "D"
      QC_FROM_U1_PE : Bool;   // QUALITY CHECK FROM UNIT 1 - PART "E"
      SPARE_14_7 : Bool;
      ANY_QC_PART_U2_PA : Bool;   // ANY PART TO QUALITY CHECK FROM UNIT 2
      ALL_QC_PART_U2_PA : Bool;   // ALL PARTS TO QUALITY CHECK FROM UNIT 2
      QC_FROM_U2_PA : Bool;   // QUALITY CHECK FROM UNIT 2 - PART "A"
      QC_FROM_U2_PB : Bool;   // QUALITY CHECK FROM UNIT 2 - PART "B"
      QC_FROM_U2_PC : Bool;   // QUALITY CHECK FROM UNIT 2 - PART "C"
      QC_FROM_U2_PD : Bool;   // QUALITY CHECK FROM UNIT 2 - PART "D"
      QC_FROM_U2_PE : Bool;   // QUALITY CHECK FROM UNIT 2 - PART "E"
      SPARE_15_7 : Bool;
      SPARE_16_0 : Byte;
      SPARE_17_0 : Byte;
      SPARE_18_0 : Byte;
      SPARE_19_0 : Byte;
   END_STRUCT;
END_TYPE

TYPE "MACHINE ALARM"
// stored: IsFailsafeCompliant false
   STRUCT
      IS_ALARMS : Bool;   // IMMEDIATE STOP ALARMS
      RHP_ALARMS : Bool;   // RETURN HOME POSITION ALARMS
      SEOC_ALARMS : Bool;   // STOP END OF CYCLE ALARMS
      IS_WARNING : Bool;   // IMMEDIATE STOP WARNING / IMMEDIATE STOP WARNINGS
      RHP_WARNING : Bool;   // RETURN HOME POSITION WARNING / RETURN HOME POSITION WARNINGS
      SEOC_WARNING : Bool;   // STOP END OF CYCLE WARNING / STOP END OF CYCLE WARNINGS
      WARNING : Bool;   // WARNING / WARNINGS
      HELP : Bool;   // HELP
      aux1_2 : Bool;   // aux1_2
      aux1_3 : Bool;   // aux1_3
      aux1_4 : Bool;   // aux1_4
      aux1_5 : Bool;   // aux1_5
      RHP_DONE_PULSE : Bool;   // RETURN HOME POSITION DONE PULSE
      RHP_DONE : Bool;   // RETURN HOME POSITION DONE
      ALARM : Bool;   // FAULT / ALARM
      RESET_ALL_SEQUENCES : Bool;   // RESET ALL SEQUENCES
      RESET_LOCAL_SEQUENCES : Bool;   // RESET LOCAL SEQUENCES
      RESET_STOP_WARNING : Bool;   // RESET STOP WARNING / RESET STOP WARNINGS
      ALARM_DECODING : DInt;   // FAULT DECODING / ALARMS DECODING
      WARNING_DECODING : DInt;   // WARNING DECODING / WARNINGS DECODING
      HELP_DECODING : DInt;   // HELP DECODING
   END_STRUCT;
END_TYPE

TYPE "UNIT ALARM"
// stored: IsFailsafeCompliant false
   STRUCT
      IS_ALARMS : Bool;   // IMMEDIATE STOP ALARMS
      IS_SEOC_ALARMS : Bool;   // IMMEDIATE STOP & STOP END OF CYCLE ALARMS / IMMEDIATE STOP AND STOP END OF CYCLE ALARMS
      RHP_ALARMS : Bool;   // RETURN HOME POSITION ALARMS
      RHP_SEOC_ALARMS : Bool;   // RETURN HOME POSITION & STOP END OF CYCLE ALARMS / RETURN HOME POSITION AND STOP END OF CYCLE ALARMS
      SEOC_ALARMS : Bool;   // STOP END OF CYCLE ALARMS
      IS_WARNING : Bool;   // IMMEDIATE STOP WARNING / IMMEDIATE STOP WARNINGS
      RHP_WARNING : Bool;   // RETURN HOME POSITION WARNING / RETURN HOME POSITION WARNINGS
      SEOC_WARNING : Bool;   // STOP END OF CYCLE WARNING / STOP END OF CYCLE WARNINGS
      WARNING : Bool;   // WARNING / WARNINGS
      HELP : Bool;   // HELP
      ALARM : Bool;   // ALARM
      WARNING_STOP : Bool;   // WARNING STOP
      RESET_ALL_SEQUENCES : Bool;   // RESET ALL SEQUENCES
      RESET_LOCAL_SEQUENCES : Bool;   // RESET LOCAL SEQUENCES
      MASK_IS : Bool;   // MASK IMMEDIATE STOP
      MASK_IS_SEOC : Bool;   // MASK IMMEDIATE STOP & STOP END OF CYCLE / MASK IMMEDIATE STOP AND STOP END OF CYCLE
      MASK_RHP : Bool;   // MASK RETURN HOME POSITION
      MASK_RHP_SEOC : Bool;   // MASK RETURN HOME POSITION & STOP END OF CYCLE / MASK RETURN HOME POSITION AND STOP END OF CYCLE
      MASK_SEOC : Bool;   // MASK STOP END OF CYCLE
      MASK_IS_WARNING : Bool;   // MASK IMMEDIATE STOP WARNING
      MASK_RHP_WARNING : Bool;   // MASK RETURN HOME POSITIONS WARNING
      MASK_SEOC_WARNING : Bool;   // MASK STOP END OF CYCLE WARNING
      MASK_WARNING : Bool;   // MASK WARNING
      MASK_HELP : Bool;   // MASK HELP
      AUX_IS : Bool;   // AUXILIARY IMMEDIATE STOP ALARMS
      AUX_IS_SEOC : Bool;   // AUXILIARY IMMEDIATE STOP & STOP END OF CYCLE ALARMS / AUXILIARY IMMEDIATE STOP AND STOP END OF CYCLE ALARMS
      AUX_RHP : Bool;   // AUXILIARY RETURN HOME POSITION ALARMS
      AUX_RHP_SEOC : Bool;   // AUXILIARY RETURN HOME POSITION & STOP END OF CYCLE ALARMS / AUXILIARY RETURN HOME POSITION AND STOP END OF CYCLE ALARMS
      AUX_SEOC : Bool;   // AUXILIARY STOP END OF CYCLE ALARMS
      AUX_IS_WARNING : Bool;   // AUXILIARY IMMEDIATE STOP WARNING / AUXILIARY IMMEDIATE STOP WARNINGS
      AUX_RHP_WARNING : Bool;   // AUXILIARY RETURN HOME POSITION WARNING / AUXILIARY RETURN HOME POSITION WARNINGS
      AUX_SEOC_WARNING : Bool;   // AUXILIARY STOP END OF CYCLE WARNING / AUXILIARY STOP END OF CYCLE WARNINGS
      AUX_WARNING : Bool;   // AUXILIARY WARNING / AUXILIARY WARNINGS
      AUX_HELP : Bool;   // AUXILIARY HELP
   END_STRUCT;
END_TYPE

TYPE "AXIS_SAFETY_IN"
// stored: IsFailsafeCompliant true
   STRUCT
      STO_Active : Bool;   // SAFE TORQUE OFF ACTIVE
      SS1_Active : Bool;   // SAFE STOP 1 ACTIVE
      SS2_Active : Bool;   // SAFE STOP 2 ACTIVE
      SOS_Active : Bool;   // SAFE OPERATING STOP ACTIVE
      SLS_Active : Bool;   // SAFE LIMITED SPEED ACTIVE
      Reserved_Input_1 : Bool;
      SLP_Active : Bool;   // SAFETY LOGIC PROGRAMME ACTIVE
      Int_Event_Active : Bool;   // INTERNAL EVENT ACTIVE
      Reserved_Input_2 : Bool;
      SLS_BIT_0_ACTIVE : Bool;   // SAFE LIMITED SPEED BIT 0 ACTIVE
      SLS_BIT_1_ACTIVE : Bool;   // SAFE LIMITED SPEED BIT 1 ACTIVE
      Reserved_Input_3 : Bool;
      SDI_POS_ACTIVE : Bool;   // SAFE DIRECTION POSITIVE ACTIVE
      SDI_NEG_ACTIVE : Bool;   // SAFE DIRECTION NEGATIVE ACTIVE
      Reserved_Input_4 : Bool;
      "SSM_n<nx" : Bool;   // SAFE SPEED MONITOR N<NX
      Reserved_Input_5 : Bool;
      Reserved_Input_6 : Bool;
      Reserved_Input_7 : Bool;
      SLP_RANGE_ACTIVE : Bool;   // SAFETY LOGIC PROGRAMME RANGE ACTIVE
      Reserved_Input_8 : Bool;
      Reserved_Input_9 : Bool;
      SAFE_POS_VALID : Bool;   // SAFE POSITION VALID
      SAFELY_REFERENCED : Bool;   // SAFELY REFERENCED
      "F-DI_0" : Bool;
      "F-DI_1" : Bool;
      "F-DI_2" : Bool;
      SS2E_ESR : Bool;   // SAFE STOP 2 EXTENDED ESR
      SS2E_ACTIVE : Bool;   // SAFE STOP 2 EXTENDED ACTIVE
      SOS_SELECTED : Bool;   // SAFE OPERATING STOP SELECTED
      SLP_UPPER_LIMIT : Bool;   // SAFETY LOGIC PROGRAMME UPPER LIMIT
      SLP_LOWER_LIMIT : Bool;   // SAFETY LOGIC PROGRAMME LOWER LIMIT
   END_STRUCT;
END_TYPE

TYPE "AXIS_SAFETY_OUT"
// stored: IsFailsafeCompliant true
   STRUCT
      Deselect_STO : Bool;   // DESELECT SAFE TORQUE OFF
      Deselect_SS1 : Bool;   // DESELECT SAFE STOP 1
      Deselect_SS2 : Bool;   // DESELECT SAFE STOP 2
      Deselect_SOS : Bool;   // DESELECT SAFE OPERATING STOP
      Deselect_SLS : Bool;   // DESELECT SAFE LIMITED SPEED
      Reserved_Out_1 : Bool;
      Deselect_SLP : Bool;   // DESELECT SAFETY LOGIC PROGRAMME
      Ack_Inc_Event : Bool;   // ACKNOWLEDGE INTERNAL EVENT ACTIVE
      Reserved_Out_2 : Bool;
      Select_SLS_bit_0 : Bool;   // SELECT SAFE LIMITED SPEED BIT 0
      Select_SLS_bit_1 : Bool;   // SELECT SAFE LIMITED SPEED BIT 1
      Reserved_Out_3 : Bool;
      Deselect_SDI_Pos : Bool;   // DESELECT SAFE DIRECTION POSITIVE
      Deselect_SDI_Neg : Bool;   // DESELECT SAFE DIRECTION NEGATIVE
      Reserved_Out_4 : Bool;
      Reserved_Out_5 : Bool;
      Reserved_Out_6 : Bool;
      Reserved_Out_7 : Bool;
      Reserved_Out_8 : Bool;
      Select_SPL_range : Bool;   // SELECT SAFETY LOGIC PROGRAMME RANGE
      Reserved_Out_9 : Bool;
      Reserved_Out_10 : Bool;
      Reserved_Out_11 : Bool;
      Des_Safe_Cam : Bool;   // DESELECT SAFETY CAMS
      Select_Gear_bit_0 : Bool;   // SELECT GEAR BIT 0
      Select_Gear_bit_1 : Bool;   // SELECT GEAR BIT 1
      Select_Gear_bit_2 : Bool;   // SELECT GEAR BIT 2
      Deselect_Gear_Sw : Bool;   // DESELECT GEAR SW
      Deselect_SS2E : Bool;   // DESELECT SAFE STOP 2 EXTENDED
      Deselect_SS2ESR : Bool;   // DESELECT SAFE STOP 2 EXTENDED ESR
      Reserved_Out_14 : Bool;   // DESELECT
      Reserved_Out_15 : Bool;   // DESELECT
      SLS1_Limit : Word;   // SAFELY LIMITED SPEED 1 LIMIT
   END_STRUCT;
END_TYPE

TYPE "SAFETY_GROUP"
// stored: IsFailsafeCompliant true
   STRUCT
      STO_Deactivate : Bool;   // SAFE TORQUE OFF DEACTIVATE
      SS1_Deactivate : Bool;   // SAFE STOP 1 DEACTIVATE
      SS2_Deactivate : Bool;   // SAFE STOP 2 DEACTIVATE
      SS2E_Deactivate : Bool;   // SAFE STOP 2 EXTENDED DEACTIVATE
      SOS_Deactivate : Bool;   // SAFE OPERATING STOP DEACTIVATE
      SLS_Deactivate : Bool;   // SAFE LIMITED SPEED DEACTIVATE
      SLS_BIT0 : Bool;   // SAFE LIMITED SPEED BIT 0
      SLS_BIT1 : Bool;   // SAFE LIMITED SPEED BIT 1
   END_STRUCT;
END_TYPE

TYPE "HOPPER"
// stored: IsFailsafeCompliant false
   STRUCT
      PRESSURIZE_PROP_GAS_VALVE_F : Int;   // PRESSURIZE PROPORTIONAL GAS VALVE FEEDBACK
      PRESSURIZE_GAS_VALVE : Bool;   // HOPPER PRESSURIZE GAS VALVE STATUS (CLOSED = 0 / OPEN = 1)
      RELIEF_GAS_VALVE : Bool;   // HOPPER RELIEF GAS VALVE STATUS (CLOSED = 0 / OPEN = 1)
      HIGH_LEVEL : Bool;   // HOPPER HIGH LEVEL SENSOR STATUS (LEVEL NOT REACHED = 0 / LEVEL REACHED= 1)
      LOW_LEVEL : Bool;   // HOPPER LOW LEVEL SENSOR STATUS (LEVEL NOT REACHED = 0 / LEVEL REACHED= 1)
      MAX_WEIGHT_SETPOINT : Real;   // MAX WEIGHT SETPOINT (kg)
      TOTAL_WEIGHT : Real;   // TOTAL WEIGHT (kg)
      HOPPER_WEIGHT_SETPOINT : Real;   // HOPPER HMI SET WEIGHT (kg)
      POWDER_WEIGHT : Real;   // POWDER WEIGHT (kg)
      UPPER_JACKET_TEMPERATURE : Real;   // HOPPER UPPER JACKET TEMPERATURE VALUE (ºC)
      UPPER_JACKET_TEMPERATURE_SETPOINT : Real;   // HOPPER UPPER JACKET TEMPERATURE SETPOINT VALUE (ºC)
      LOWER_JACKET_TEMPERATURE : Real;   // HOPPER LOWER JACKET TEMPERATURE VALUE (ºC)
      LOWER_JACKET_TEMPERATURE_SETPOINT : Real;   // HOPPER LOWER JACKET TEMPERATURE SETPOINT VALUE (ºC)
      HOPPER_PRESSURE : Real;   // HOPPER COVER PRESSURE VALUE (Bar)
      HOPPER_PRESSURE_SETPOINT : Real;   // HOPPER COVER PRESSURE SETPOINT VALUE (Bar)
      STIRRER_CURRENT : DInt;   // HOPPER STIRRER CURRENT VALUE (mA)
      STIRRER_SPEED : DInt;   // HOPPER STIRRER SPEED VALUE (RPM or %)
      STIRRER_SPEED_SETPOINT : DInt;   // HOPPER STIRRER SPEED SETPOINT VALUE (RPM or %)
      TRANSFER_POWDER_VALVE : Bool;   // HOPPER TRANSFER POWDER VALVE STATUS (CLOSED = 0 / OPEN = 1)
      CLEANING_AIR_VALVE : Bool;
      LOAD_FEEDER_SEQ : Bool;
      POWDER_FLOW : Array[1..20] of "MEDICOAT_TIME_STAMP";   // HOPPER POWDER FLOW VALUE (Raw)
   END_STRUCT;
END_TYPE

TYPE "MEDICOAT_TIME_STAMP"
// stored: IsFailsafeCompliant false
   STRUCT
      VALUE : Int;
      TIME_STAMP : DTL;
   END_STRUCT;
END_TYPE

TYPE "POWDER_FEEDER_LINE"
// stored: IsFailsafeCompliant false
   STRUCT
      HOPPER : Struct
         PRESSURE : Real;   // POWDER FEEDER HOPPER PRESSURE VALUE (Bar)
         TEMPERATURE : Real;   // POWDER FEEDER HOPPER TEMPERATURE VALUE (ºC)
         TEMPERATURE_SETPOINT : Real;   // POWDER FEEDER HOPPER TEMPERATURE SETPOINT VALUE (ºC)
         STIRRER_CURRENT : Int;   // POWDER FEEDER HOPPER STIRRER CURREN VALUE (mA)
         STIRRER_SPEED : Real;   // POWDER FEEDER HOPPER STIRRER SPEED VALUE (RPM or %)
         STIRRER_SPEED_SETPOINT : Real;   // POWDER FEEDER HOPPER STIRRER SPEED SETPOINT VALUE (RPM or %)
      END_STRUCT;
      DISC : Struct
         CURRENT : Int;   // POWDER FEEDER DISC CURRENT VALUE (mA)
         SPEED : Real;   // POWDER FEEDER DISC SPEED VALUE (RPM or %)
         SPEED_SETPOINT : Real;   // POWDER FEEDER DISC SPEED SET POINT VALUE (RPM or %)
      END_STRUCT;
      CARRIER_GAS : Struct
         PRESSURE : Real;   // POWDER FEEDER CARRIER GAS PRESSURE VALUE (Bar)
         FLOW : Real;   // POWDER FEEDER CARRIER GAS FLOW VALUE (NLPM)
         FLOW_SETPOINT : Real;   // POWDER FEEDER CARRIER GAS FLOW SETPOINT VALUE (NLPM)
      END_STRUCT;
      POWDER_FLOW : Array[1..20] of "MEDICOAT_TIME_STAMP";   // POWDER FEEDER POWDER FLOW VALUE (Raw)
      POWDER_TYPE { ExternalWritable := 'False'} : Struct
         MANUFACTURER { ExternalWritable := 'False'} : Array[0..20] of Char;   // POWDER TYPE: MANUFACTURER IDENTIFICATION
         REFERENCE { ExternalWritable := 'False'} : Array[0..20] of Char;   // POWDER TYPE: POWDER REFERENCE
         BATCH_NUMBER { ExternalWritable := 'False'} : Array[0..20] of Char;   // POWDER TYPE: POWDER BATCH NUMBER
         CONTAINER_ID { ExternalWritable := 'False'} : Array[0..20] of Char;   // POWDER TYPE: POWDER CONTAINER IDENTIFICATION
         HUMIDITY { ExternalWritable := 'False'} : Real;   // POWDER TYPE: HUMIDITY VALUE (¿?¿?¿?¿?)
         GRANULOMETRY { ExternalWritable := 'False'} : Real;   // POWDER TYPE: GRANULOMETRY VALUE (¿?¿?¿?¿?)
         POROSITY { ExternalWritable := 'False'} : Real;   // POWDER TYPE: POROSITY VALUE (¿?¿?¿?¿?)
      END_STRUCT;
      STATUS : Struct
         RUNNING : Bool;
      END_STRUCT;
   END_STRUCT;
END_TYPE

TYPE "POWDER FEEDER INTERLOCK INPUT"
// stored: IsFailsafeCompliant false
   STRUCT
      i_uiOperationMode_Line1 : Word;   // Current Line Operation Mode 0 = Stand Alone, 1 = On Off Remote 2 = UDP, 3 = Profibus, 5 = Device Net / current line operation mode 0 = Standalone, 1 = OnOffRemote 2 = UDP, 3 = Profibus, 4 = ProfiNet, 5 = DeviceNet
      i_uiOperationMode_Line2 : Word;   // Current Line Operation Mode 0 = Stand Alone, 1 = On Off Remote 2 = UDP, 3 = Profibus, 5 = Device Net / current line operation mode 0 = Standalone, 1 = OnOffRemote 2 = UDP, 3 = Profibus, 4 = ProfiNet, 5 = DeviceNet
      i_uiFeederState_Line1 : Word;   // Current Feeder Line StateCG_Feedfun_Disabled=0, Cg_Ready_Start=1,Cg_Wait_To_Eestablish=2, Feedfunc_Ready_Start=3,Feedfun_Running=4, Feedfun_Wait_To_Zero=5 / current feeder line state CG_FEEDFUN_DISABLED=0, CG_READY_START=1, CG_WAIT_TO_ESTABLISH=2, FEEDFUNC_READY_START=3, FEEDFUN_RUNNING=4, FEEDFUN_WAIT_TO_ZERO=5
      i_uiFeederState_Line2 : Word;   // Current Feeder Line StateCG_Feedfun_Disabled=0, Cg_Ready_Start=1,Cg_Wait_To_Establish=2, Feedfunc_Ready_Start=3,Feedfun_Running=4, Feedfun_Wait_To_Zero=5 / current feeder line state CG_FEEDFUN_DISABLED=0, CG_READY_START=1, CG_WAIT_TO_ESTABLISH=2, FEEDFUNC_READY_START=3, FEEDFUN_RUNNING=4, FEEDFUN_WAIT_TO_ZERO=5
      i_fOperationModeMatched_Line1 : Bool;   // O_UiOperationMode Is Equal To Feeder Line Operation Mode / o_uiOperationMode is equal to feeder line operation mode
      i_fOperationModeMatched_Line2 : Bool;   // O_UiOperationMode Is Equal To Feeder Line Operation Mode / o_uiOperationMode is equal to feeder line operation mode
      i_fFeedingMode_Line1 : Bool;   // 0 = Volumetric (For Twin 150 Always Volumetric) 1 = Gravimetric / 0 = volumetric (for Twin 150 always volumetric), 1 = gravimetric
      i_fFeedingMode_Line2 : Bool;   // 0 = Volumetric (For Twin 150 Always Volumetric) 1 = Gravimetric / 0 = volumetric (for Twin 150 always volumetric), 1 = gravimetric
      i_fFeederReady_Line1 : Bool;   // No Shutdown Present / No shutdown present
      i_fFeederReady_Line2 : Bool;   // No Shutdown Present / No shutdown present
      i_fTareDone_Line1 : Bool;   // N/a For Twin 150 / n/a for Twin 150
      i_fTareDone_Line2 : Bool;   // N/a For Twin 150 / n/a for Twin 150
      i_fCalibDone_Line1 : Bool;   // N/a For Twin 150 / n/a for Twin 150
      i_fCalibDone_Line2 : Bool;   // N/a For Twin 150 / n/a for Twin 150
      i_fCarrierGasSelected_Line1 : Bool;   // 0 = Argon Selected, 1 = Nitrogen Selected / 0 = Argon selected, 1 = Nitrogen selected
      i_fCarrierGasSelected_Line2 : Bool;   // 0 = Argon Selected, 1 = Nitrogen Selected / 0 = Argon selected, 1 = Nitrogen selected
      i_fUnitSelected_Line1 : Bool;   // 0 = Metric Units, 1 = SI / 0 = metric units, 1 = SI
      i_fUnitSelected_Line2 : Bool;   // 0 = Metric Units, 1 = SI / 0 = metric units, 1 = SI
      i_fPowderLineClogged_Line1 : Bool;   // 0 = Line Not Clogged, 1 = Line Is Clogged (Overpressure) / 0 = line not clogged, 1 = line is clogged (overpressure)
      i_fPowderLineClogged_Line2 : Bool;   // 0 = Line Not Clogged, 1 = Line Is Clogged (Overpressure) / 0 = line not clogged, 1 = line is clogged (overpressure)
      i_fShutdownFromPf_Line1 : Bool;   // 0 = No Shutdown Present, 1 = Shutdown Present For Feeder Line / 0 = no shutdown present, 1 = shutdown present for feeder line
      i_fShutdownFromPf_Line2 : Bool;   // 0 = No Shutdown Present, 1 = Shutdown Present For Feeder Line / 0 = no shutdown present, 1 = shutdown present for feeder line
      i_fWarningFromPF_Line1 : Bool;   // 0 = No Warning Present, 1 = Warning Present For Feeder Line / 0 = no warning present, 1 = warning present for feeder line
      i_fWarningFromPF_Line2 : Bool;   // 0 = No Warning Present, 1 = Warning Present For Feeder Line / 0 = no warning present, 1 = warning present for feeder line
      i_fDiskStatus_Line1 : Bool;   // 0 = Disk Motor Not Ready, 1 = Disk Motor Plugged In And Ready / 0 = disk motor not ready, 1 = disk motor plugged in and ready
      i_fDiskStatus_Line2 : Bool;   // 0 = Disk Motor Not Ready, 1 = Disk Motor Plugged In And Ready / 0 = disk motor not ready, 1 = disk motor plugged in and ready
      i_fStirrerStatus_Line1 : Bool;   // 0 = Stirrer Motor Not Ready, 1 = Stirrer Is Plugged In And Ready / 0 = stirrer motor not ready, 1 = stirrer is plugged in and ready
      i_fStirrerStatus_Line2 : Bool;   // 0 = Stirrer Motor Not Ready, 1 = Stirrer Is Plugged In And Ready / 0 = stirrer motor not ready, 1 = stirrer is plugged in and ready
      i_fCarriergasStatus_Line1 : Bool;   // 0 = Carrier Gas Is Off, 1 = Carrier Gas Is Running / 0 = carriergas is off, 1 = carriergas is running
      i_fCarriergasStatus_Line2 : Bool;   // 0 = Carrier Gas Is Off, 1 = Carrier Gas Is Running / 0 = carriergas is off, 1 = carriergas is running
      i_fCommunicationOK_Line1 : Bool;   // 1 = Communication Running / 1 = Communication running
      i_fCommunicationOK_Line2 : Bool;   // 1 = Communication Running / 1 = Communication running
      i_fCarriergasLeLL_Line1 : Bool;   // 0 = Carrier Gas Flow > LL Limit, 1 = Carrier Gas Flow < LL Limit / 0 = carriergas flow > LL limit, 1 = carriergas flow < LL limit
      i_fCarriergasLeLL_Line2 : Bool;   // 0 = Carrier Gas Flow > LL Limit, 1 = Carrier Gas Flow < LL Limit / 0 = carriergas flow > LL limit, 1 = carriergas flow < LL limit
      i_fDiskSpeedLeLL_Line1 : Bool;   // 0 = Disk Speed > LL Limit, 1 = Disk Speed < LL Limit / 0 = disk speed > LL limit, 1 = disk speed < LL limit
      i_fDiskSpeedLeLL_Line2 : Bool;   // 0 = Disk Speed > LL Limit, 1 = Disk Speed < LL Limit / 0 = disk speed > LL limit, 1 = disk speed < LL limit
      i_fStirrerSpeedLeLL_Line1 : Bool;   // 0 = Stirrer Speed > LL Limit, 1 = Stirrer Speed < LL Limit / 0 = stirrer speed > LL limit, 1 = stirrer speed < LL limit
      i_fStirrerSpeedLeLL_Line2 : Bool;   // 0 = Stirrer Speed > LL Limit, 1 = Stirrer Speed < LL Limit / 0 = stirrer speed > LL limit, 1 = stirrer speed < LL limit
      i_fFeedrateLeLL_Line1 : Bool;   // N/a For Twin 150 / n/a for Twin 150
      i_fFeedrateLeLL_Line2 : Bool;   // N/a For Twin 150 / n/a for Twin 150
      i_fPowderLevelLeLL_Line1 : Bool;   // N/a For Twin 150 / n/a for Twin 150
      i_fPowderLevelLeLL_Line2 : Bool;   // N/a For Twin 150 / n/a for Twin 150
      i_fCarriergasLeL_Line1 : Bool;   // 0 = Carrier Gas Flow > L Limit, 1 = Carrier Gas Flow < L Limit / 0 = carriergas flow > L limit, 1 = carriergas flow < L limit
      i_fCarriergasLeL_Line2 : Bool;   // 0 = Carrier Gas Flow > L Limit, 1 = Carrier Gas Flow < L Limit / 0 = carriergas flow > L limit, 1 = carriergas flow < L limit
      i_fDiskSpeedLeL_Line1 : Bool;   // 0 = Disk Speed > L Limit, 1 = Disk Speed < L Limit / 0 = disk speed > L limit, 1 = disk speed < L limit
      i_fDiskSpeedLeL_Line2 : Bool;   // 0 = Disk Speed > L Limit, 1 = Disk Speed < L Limit / 0 = disk speed > L limit, 1 = disk speed < L limit
      i_fStirrerSpeedLeL_Line1 : Bool;   // 0 = Stirrer Speed > L Limit, 1 = Stirrer Speed < L Limit / 0 = Stirrer speed > L limit, 1 = Stirrer speed < L limit
      i_fStirrerSpeedLeL_Line2 : Bool;   // 0 = Stirrer Speed > L Limit, 1 = Stirrer Speed < L Limit / 0 = Stirrer speed > L limit, 1 = Stirrer speed < L limit
      i_fFeedrateLeL_Line1 : Bool;   // N/a For Twin 150 / n/a for Twin 150
      i_fFeedrateLeL_Line2 : Bool;   // N/a For Twin 150 / n/a for Twin 150
      i_fPowderLevelLeL_Line1 : Bool;   // N/a For Twin 150 / n/a for Twin 150
      i_fPowderLevelLeL_Line2 : Bool;   // N/a For Twin 150 / n/a for Twin 150
      i_fCarriergasGrH_Line1 : Bool;   // 0 = Carrier Gas Flow < H Limit, 1 = Carrier Gas Flow > H Limit / 0 = carriergas flow < H limit, 1 = carriergas flow > H limit
      i_fCarriergasGrH_Line2 : Bool;   // 0 = Carrier Gas Flow < H Limit, 1 = Carrier Gas Flow > H Limit / 0 = carriergas flow < H limit, 1 = carriergas flow > H limit
      i_fDiskSpeedGrH_Line1 : Bool;   // 0 = Disk Speed < H Limit, 1 = Disk Speed > H Limit / 0 = disk speed < H limit, 1 = disk speed > H limit
      i_fDiskSpeedGrH_Line2 : Bool;   // 0 = Disk Speed < H Limit, 1 = Disk Speed > H Limit / 0 = disk speed < H limit, 1 = disk speed > H limit
      i_fStirrerSpeedGrH_Line1 : Bool;   // 0 = Stirrer Speed < H Limit, 1 = Stirrer Speed > H Limit / 0 = Stirrer speed < H limit, 1 = Stirrer speed > H limit
      i_fStirrerSpeedGrH_Line2 : Bool;   // 0 = Stirrer Speed < H Limit, 1 = Stirrer Speed > H Limit / 0 = Stirrer speed < H limit, 1 = Stirrer speed > H limit
      i_fFeedrateGrH_Line1 : Bool;   // N/a For Twin 150 / n/a for Twin 150
      i_fFeedrateGrH_Line2 : Bool;   // N/a For Twin 150 / n/a for Twin 150
      i_fCarriergasGrHH_Line1 : Bool;   // 0 = Carrier Gas Flow < HH Limit, 1 = Carriergas Flow > HH Limit / 0 = carriergas flow < HH limit, 1 = carriergas flow > HH limit
      i_fCarriergasGrHH_Line2 : Bool;   // 0 = Carrier Gas Flow < HH Limit, 1 = Carriergas Flow > HH Limit / 0 = carriergas flow < HH limit, 1 = carriergas flow > HH limit
      i_fDiskSpeedGrHH_Line1 : Bool;   // 0 = Disk Speed < HH Limit, 1 = Disk Speed > HH Limit / 0 = disk speed < HH limit, 1 = disk speed > HH limit
      i_fDiskSpeedGrHH_Line2 : Bool;   // 0 = Disk Speed < HH Limit, 1 = Disk Speed > HH Limit / 0 = disk speed < HH limit, 1 = disk speed > HH limit
      i_fStirrerSpeedGrHH_Line1 : Bool;   // 0 = Stirrer Speed < HH Limit, 1 = Stirrer Speed > HH Limit / 0 = Stirrer speed < HH limit, 1 = Stirrer speed > HH limit
      i_fStirrerSpeedGrHH_Line2 : Bool;   // 0 = Stirrer Speed < HH Limit, 1 = Stirrer Speed > HH Limit / 0 = Stirrer speed < HH limit, 1 = Stirrer speed > HH limit
      i_fHopperTempGrHH_Line1 : Bool;   // 0 = Hopper Temperature < HH Limit 110ºC, 1 = Hopper Temperature > HH Limit 110ºC / 0 = Hopper temperature < 110 °C, 1 = Hopper temperature > 110 °C
      i_fHopperTempGrHH_Line2 : Bool;   // 0 = Hopper Temperature < HH Limit 110ºC, 1 = Hopper Temperature > HH Limit 110ºC / 0 = Hopper temperature < 110 °C, 1 = Hopper temperature > 110 °C
      i_fFeedrateGrHH_Line1 : Bool;   // N/a For Twin 150 / 0 = Feedrate < HH limit, 1 = Feedrate > HH limit
      i_fFeedrateGrHH_Line2 : Bool;   // N/a For Twin 150 / 0 = Feedrate < HH limit, 1 = Feedrate > HH limit
      i_fCarriergasInletPressureTooLow_Line1 : Bool;   // 0 = Carrier Gas Pressure OK. 1 = Carriergas Pressure Too Low (Only If Pressure Switch Available) / 0 = carriergas pressure OK, 1 = carriergas pressure too low (only if pressure switch available)
      i_fCarriergasInletPressureTooLow_Line2 : Bool;   // 0 = Carrier Gas Pressure OK. 1 = Carriergas Pressure Too Low (Only If Pressure Switch Available) / 0 = carriergas pressure OK, 1 = carriergas pressure too low (only if pressure switch available)
      Spare_0 : Bool;   // Spare
      Spare_1 : Bool;   // Spare
      Spare_2 : Bool;   // Spare
      Spare_3 : Bool;   // Spare
      i_f_OptionHeatingAvailable_Line1 : Bool;   // 1 = Option Available / 1 = option available
      i_f_OptionHeatingAvailable_Line2 : Bool;   // 1 = Option Available / 1 = option available
      Spare_4 : Bool;   // Spare
      Spare_5 : Bool;   // Spare
      Spare_6 : Bool;   // Spare
      Spare_7 : Bool;   // Spare
      Spare_8 : Bool;   // Spare
      Spare_9 : Bool;   // Spare
      i_fCarrierGasType : Word;   // Spare / actual active carrier gas type: 0=Argon, 1=Nitrogen, 2=Helium, 3=Argon30
      "Actual PF Values" : Struct
         i_rCarriergasActual_Line1 : Real;   // Actual Value Carriergas Flow (NLPM) / actual value carriergas flow [NLPM]
         i_rCarriergasActual_Line2 : Real;   // Actual Value Carriergas Flow (NLPM) / actual value carriergas flow [NLPM]
         i_rDiskActual_Line1 : Real;   // Actual Value Disk Speed (%) / actual value disk speed [%]
         i_rDiskActual_Line2 : Real;   // Actual Value Disk Speed (%) / actual value disk speed [%]
         i_rStirrerActual_Line1 : Real;   // Actual Value Stirrer Speed (%) / actual value stirrer speed [%]
         i_rStirrerActual_Line2 : Real;   // Actual Value Stirrer Speed (%) / actual value stirrer speed [%]
         i_rFeedrateActual_Line1 : Real;   // N/A For Twin 150 / n/a for Twin 150
         i_rFeedrateActual_Line2 : Real;   // N/A For Twin 150 / n/a for Twin 150
         i_rHopperTempActual_Line1 : Real;   // Actual Value Hopper Temperature (ºC) / actual value hopper temperature [°C]
         i_rHopperTempActual_Line2 : Real;   // Actual Value Hopper Temperature (ºC) / actual value hopper temperature [°C]
         i_rHopperPressureActual_Line1 : Real;   // Actual Value Hopper Pressure (Bar) / actual value hopper pressure [Bar]
         i_rHopperPressureActual_Line2 : Real;   // Actual Value Hopper Pressure (Bar) / actual value hopper pressure [Bar]
         i_rWeightActual_Line1 : Real;   // N/A For Twin 150 / n/a for Twin 150
         i_rWeightActual_Line2 : Real;   // N/A For Twin 150 / n/a for Twin 150
         i_rPowderFactorActual_Line1 : Real;   // N/A For Twin 150 / n/a for Twin 150
         i_rPowderFactorActual_Line2 : Real;   // N/A For Twin 150 / n/a for Twin 150
      END_STRUCT;
   END_STRUCT;
END_TYPE

TYPE "POWDER FEEDER INTERLOCK OUTPUT"
// stored: IsFailsafeCompliant false
   STRUCT
      o_uiOperationMode : Word;   // Operation Mode 0 = Standalone, 1 = On Off Remote 2 = UDP, 3 = Profibus / operation mode 2 = UDP, 3 = Profibus, 4 = ProfiNet
      o_uiCarrierGasTypeRequest : Word;   // Spare / carrier gas selection. 0=no selection, 1=Argon, 2=Nitrogen, 3=Helium, 4=Argon30
      o_uiProductionMode : Word;   // Production Mode 0 = Off, 1 = Production / production mode 0 = OFF, 1 = Production
      Spare_Word_1 : Word;   // Spare
      o_uiSystemMode : Word;   // 0 = Plasma 1 = HVOF
      Spare_Word_2 : Word;   // Spare
      o_fAirFlowIsRunning : Bool;   // 0 = No Airflow, 1 = Airflow Present / 0 = no airflow, 1 = Airflow present
      o_fCarrierGasSelect : Bool;   // 0 = Carrier Gas Argon, 1 = Carrier Gas Nitrogen / 0 = carriergas Argon, 1 = carriergas Nitrogen
      o_fUnitSelect : Bool;   // 0 = Metric, 1 = SI / 0 = metric, 1 = SI
      Spare_0 : Bool;   // Spare
      Spare_1 : Bool;   // Spare
      Spare_2 : Bool;   // Spare
      Spare_3 : Bool;   // Spare
      Spare_4 : Bool;   // Spare
      o_fVolumetricMode_Line1 : Bool;   // 1 = Volumetric Mode On / 1 = volumetric mode on
      o_fVolumetricMode_Line2 : Bool;   // 1 = Volumetric Mode On / 1 = volumetric mode on
      o_fGravimetricMode_Line1 : Bool;   // 1 = Gravimetric Mode On n/a for Twin 150 / 1 = gravimetric mode on n/a for Twin 150
      o_fGravimetricMode_Line2 : Bool;   // 1 = Gravimetric Mode On n/a for Twin 150 / 1 = gravimetric mode on n/a for Twin 150
      o_fTareCmd_Line1 : Bool;   // N/a For Twin 150 / n/a for Twin 150
      o_fTareCmd_Line2 : Bool;   // N/a For Twin 150 / n/a for Twin 150
      Spare_5 : Bool;   // Spare
      Spare_6 : Bool;   // Spare
      o_fCalibCmd_Line1 : Bool;   // N/a For Twin 150 / n/a for Twin 150
      o_fCalibCmd_Line2 : Bool;   // N/a For Twin 150 / n/a for Twin 150
      Spare_7 : Bool;   // Spare
      Spare_8 : Bool;   // Spare
      o_fShutdownToPF_Line1 : Bool;   // 0 = Controller Doesn't Request Shutdown / 0 = controller doesn't request shutdown, 1 = controller requests shutdown
      o_fShutdownToPF_Line2 : Bool;   // 1 = Controller Requests Shutdown / 0 = controller doesn't request shutdown, 1 = controller requests shutdown
      o_fCommunicationOk_Line1 : Bool;   // Communication Is Running / Communication is running
      o_fCommunicationOk_Line2 : Bool;   // Communication Is Running / Communication is running
      o_fFeedingAllOnCmd_Line1 : Bool;   // 1 = Start Stirrer & Disk (Pos. Edge Trigger) / 1 = start stirrer & disk (pos. Edge trigger)
      o_fFeedingAllOnCmd_Line2 : Bool;   // 1 = Start Stirrer & Disk (Pos. Edge Trigger) / 1 = start stirrer & disk (pos. Edge trigger)
      o_fCarriergasOnCmd_Line1 : Bool;   // 1 = Start Carrier Gas / 1 = start carriergas (pos. Edge trigger)
      o_fCarriergasOnCmd_Line2 : Bool;   // 1 = Start Carrier Gas / 1 = start carriergas (pos. Edge trigger)
      o_fFeedingAllOffCmd_Line1 : Bool;   // 1 = Stop Stirrer & Disk / 1 = stop stirrer & disk
      o_fFeedingAllOffCmd_Line2 : Bool;   // 1 = Stop Stirrer & Disk / 1 = stop stirrer & disk
      o_fCarriergasOffCmd_Line1 : Bool;   // 1 = Stop Carrier Gas / 1 = stop carriergas
      o_fCarriergasOffCmd_Line2 : Bool;   // 1 = Stop Carrier Gas / 1 = stop carriergas
      o_fHeatingOnCmd_Line1 : Bool;   // 1 = Start Heating (Pos. Edge Trigger) / 1 = start heating (pos. Edge trigger)
      o_fHeatingOnCmd_Line2 : Bool;   // 1 = Start Heating (Pos. Edge Trigger) / 1 = start heating (pos. Edge trigger)
      o_fHeatingOffCmd_Line1 : Bool;   // 1 = Stop Heating / 1 = stop heating
      o_fHeatingOffCmd_Line2 : Bool;   // 1 = Stop Heating / 1 = stop heating
      Spare_9 : Bool;   // Spare
      Spare_10 : Bool;   // Spare
      Spare_11 : Bool;   // Spare
      Spare_12 : Bool;   // Spare
      Spare_Byte_0 : Byte;   // Spare
      Spare_Byte_1 : Byte;   // Spare
      Spare_Byte_2 : Byte;   // Spare
      "PF Setpoints, Warnings and Alarms" : Struct
         o_rCarriergasNominal_Line1 : Real;   // Carrier Gas Setpoint [NLPM] (0..16 NLPM) / carriergas setpoint [NLPM] (0..16 NLPM)
         o_rCarriergasNominal_Line2 : Real;   // Carrier Gas Setpoint [NLPM] (0..16 NLPM) / carriergas setpoint [NLPM] (0..16 NLPM)
         o_rDiskSpeedNominal_Line1 : Real;   // Disk Speed Setpoint [%] (0..100 %) / Disk speed setpoint [%] (0..100 %)
         o_rDiskSpeedNominal_Line2 : Real;   // Disk Speed Setpoint [%] (0..100 %) / Disk speed setpoint [%] (0..100 %)
         o_rStirrerSpeedNominal_Line1 : Real;   // Stirrer Speed Setpoint [%] (30 - 100%) / Stirrer speed setpoint [%] (30 - 100%)
         o_rStirrerSpeedNominal_Line2 : Real;   // Stirrer Speed Setpoint [%] (30 - 100%) / Stirrer speed setpoint [%] (30 - 100%)
         o_rFeedrateNominal_Line1 : Real;   // N/a For Twin 150 / n/a for Twin 150
         o_rFeedrateNominal_Line2 : Real;   // N/a For Twin 150 / n/a for Twin 150
         o_rHopperTempNominal_Line1 : Real;   // Hopper Temperature Setpoint [°C] (n/a for Twin 150 R1.0) / Hopper temperature setpoint [°C]
         o_rHopperTempNominal_Line2 : Real;   // Hopper Temperature Setpoint [°C] (n/a for Twin 150 R1.0) / Hopper temperature setpoint [°C]
         o_rLoadcellCalibrationNominal_Line1 : Real;   // N/a For Twin 150 / n/a for Twin 150
         o_rLoadcellCalibrationNominal_Line2 : Real;   // N/a For Twin 150 / n/a for Twin 150
         o_rPowderFactorNominal_Line1 : Real;   // N/a For Twin 150 / n/a for Twin 150
         o_rPowderFactorNominal_Line2 : Real;   // N/a For Twin 150 / n/a for Twin 150
         o_rLLlimitCarriergas_Line1 : Real;   // Carrier Gas Flow LL Limit [NLPM] (Absolute Value) / carriergas flow LL limit [NLPM] (absolute value)
         o_rLLlimitCarriergas_Line2 : Real;   // Carrier Gas Flow LL Limit [NLPM] (Absolute Value) / carriergas flow LL limit [NLPM] (absolute value)
         o_rLLlimitDiskSpeedNominal_Line1 : Real;   // Disk Speed LL Limit [%] (Absolute Value) / Disk speed LL limit [%] (absolute value)
         o_rLLlimitDiskSpeedNominal_Line2 : Real;   // Disk Speed LL Limit [%] (Absolute Value) / Disk speed LL limit [%] (absolute value)
         o_rLLlimitStirrerSpeedNominal_Line1 : Real;   // Stirrer Speed LL Limit [%] (Absolute Value) / Stirrer speed LL limit [%] (absolute value)
         o_rLLlimitStirrerSpeedNominal_Line2 : Real;   // Stirrer Speed LL Limit [%] (Absolute Value) / Stirrer speed LL limit [%] (absolute value)
         o_rLLlimitFeedRateNominal_Line1 : Real;   // N/a For Twin 150 / n/a for Twin 150
         o_rLLlimitFeedRateNominal_Line2 : Real;   // N/a For Twin 150 / n/a for Twin 150
         o_rLlimitCarriergas_Line1 : Real;   // Carrier Gas L Limit [NLPM] (Absolute Value) / carriergas L limit [NLPM] (absolute value)
         o_rLlimitCarriergas_Line2 : Real;   // Carrier Gas L Limit [NLPM] (Absolute Value) / carriergas L limit [NLPM] (absolute value)
         o_rLlimitDiskSpeedNominal_Line1 : Real;   // Disk Speed L Limit [%] (Absolute Value) / Disk speed L limit [%] (absolute value)
         o_rLlimitDiskSpeedNominal_Line2 : Real;   // Disk Speed L Limit [%] (Absolute Value) / Disk speed L limit [%] (absolute value)
         o_rLlimitStirrerSpeedNominal_Line1 : Real;   // Stirrer Speed L Limit [%] (Absolute Value) / Stirrer speed L limit [%] (absolute value)
         o_rLlimitStirrerSpeedNominal_Line2 : Real;   // Stirrer Speed L Limit [%] (Absolute Value) / Stirrer speed L limit [%] (absolute value)
         o_rLlimitFeedRateNominal_Line1 : Real;   // N/a For Twin 150 / n/a for Twin 150
         o_rLlimitFeedRateNominal_Line2 : Real;   // N/a For Twin 150 / n/a for Twin 150
         o_rHlimitCarriergas_Line1 : Real;   // Carrier Gas H Limit [NLPM] (Absolute Value) / Carriergas H limit [NLPM] (absolute value)
         o_rHlimitCarriergas_Line2 : Real;   // Carrier Gas H Limit [NLPM] (Absolute Value) / Carriergas H limit [NLPM] (absolute value)
         o_rHlimitDiskSpeedNominal_Line1 : Real;   // Disk Speed H Limit [%] (Absolute Value) / Disk speed H limit [%] (absolute value)
         o_rHlimitDiskSpeedNominal_Line2 : Real;   // Disk Speed H Limit [%] (Absolute Value) / Disk speed H limit [%] (absolute value)
         o_rHlimitStirrerSpeedNominal_Line1 : Real;   // Stirrer Speed H Limit [%] (Absolute Value) / Stirrer speed H limit [%] (absolute value)
         o_rHlimitStirrerSpeedNominal_Line2 : Real;   // Stirrer Speed H Limit [%] (Absolute Value) / Stirrer speed H limit [%] (absolute value)
         o_rHlimitFeedRateNominal_Line1 : Real;   // N/a For Twin 150 / n/a for Twin 150
         o_rHlimitFeedRateNominal_Line2 : Real;   // N/a For Twin 150 / n/a for Twin 150
         o_rHHlimitCarriergas_Line1 : Real;   // Carrier Gas HH Limit [NLPM] (Absolute Value) / Carriergas HH limit [NLPM] (absolute value)
         o_rHHlimitCarriergas_Line2 : Real;   // Carrier Gas HH Limit [NLPM] (Absolute Value) / Carriergas HH limit [NLPM] (absolute value)
         o_rHHlimitDiskSpeedNominal_Line1 : Real;   // Disk Speed HH Limit [%] (Absolute Value) / Disk speed HH limit [%] (absolute value)
         o_rHHlimitDiskSpeedNominal_Line2 : Real;   // Disk Speed HH Limit [%] (Absolute Value) / Disk speed HH limit [%] (absolute value)
         o_rHHlimitStirrerSpeedNominal_Line1 : Real;   // Stirrer Speed HH Limit [%] (Absolute Value) / Stirrer speed HH limit [%] (absolute value)
         o_rHHlimitStirrerSpeedNominal_Line2 : Real;   // Stirrer Speed HH Limit [%] (Absolute Value) / Stirrer speed HH limit [%] (absolute value)
         o_rHHlimitFeedRateNominal_Line1 : Real;   // N/a For Twin 150 / n/a for Twin 150
         o_rHHlimitFeedRateNominal_Line2 : Real;   // N/a For Twin 150 / n/a for Twin 150
         o_rHHlimitHopperTempNominal_Line1 : Real;   // Hopper Temperature HH Limit (ºC), (Absolute Value, N/a For Twin 150 R1.0) / Hopper temperature HH limit [°C] (absolute value, n/a for Twin 150)
         o_rHHlimitHopperTempNominal_Line2 : Real;   // Hopper Temperature HH Limit (ºC), (Absolute Value, N/a For Twin 150 R1.0) / Hopper temperature HH limit [°C] (absolute value, n/a for Twin 150)
      END_STRUCT;
   END_STRUCT;
END_TYPE

TYPE "POWDER FEEDER OERLIKON"
// stored: IsFailsafeCompliant false
   STRUCT
      Inputs : "POWDER FEEDER INTERLOCK INPUT";
      Outputs : "POWDER FEEDER INTERLOCK OUTPUT";
   END_STRUCT;
END_TYPE

TYPE "POWDER FEEDER CNC VALUES SETPOINTS"
// stored: IsFailsafeCompliant false
   STRUCT
      CarrierGasNominalLine1 : Real;
      CarrierGasNominalLine2 : Real;
      DiskSpeedNominalLine1 : Real;
      DiskSpeedNominalLine2 : Real;
      StirrerSpeedNominalLine1 : Real;
      StirrerSpeedNominalLine2 : Real;
      HopperTempNominalLine1 : Real;
      HopperTempNominalLine2 : Real;
   END_STRUCT;
END_TYPE

TYPE "POWDER FEEDER GENERAL"
// stored: IsFailsafeCompliant false
   STRUCT
      "START GENERAL CONDITIONS" : Bool;   // Start General Conditions
      "START INITIAL CONDITIONS" : Bool;   // Start Initial Conditions
      "START MANUAL REQUEST" : Bool;   // Start Manual Request
      "START AUTO REQUEST" : Bool;   // Start Auto Request
      "START GLOBAL REQUEST" : Bool;   // Start Global Request
      "START COMMAND" : Bool;   // Start Command
      START : Bool;   // Start
      "FEEDBACK ON" : Bool;   // Feedback On
      "STOP GENERAL CONDITIONS" : Bool;   // Stop General Conditions
      "STOP INITIAL CONDITIONS" : Bool;   // Stop Initial Conditions
      "STOP MANUAL REQUEST" : Bool;   // Stop Manual Request
      "STOP AUTO REQUEST" : Bool;   // Stop Auto Request
      "STOP GLOBAL REQUEST" : Bool;   // Stop Global Request
      "STOP COMMAND" : Bool;   // Stop Command
      STOP : Bool;   // Stop
      "FEEDBACK OFF" : Bool;   // Feedback Off
      "FEEDBACK ON AUX FOR HMI" : Bool;   // Feedback On Aux for HMI
      "CG FEEDFUN DISABLED LINE 1" : Bool;   // CG Feedfun Disabled Line 1
      "CG READY START LINE 1" : Bool;   // CG Ready Start Line 1
      "CG WAIT TO ESTABLISH LINE 1" : Bool;   // CG Wait To Establish Line 1
      "FEEDFUNC READY START LINE 1" : Bool;   // Feedfunc Ready Start Line 1
      "FEEDFUN RUNNING LINE 1" : Bool;   // Feedfun Running Line 1
      "FEEDFUN WAIT TO ZERO LINE 1" : Bool;   // Feedfun Wait To Zero Line 1
      "CG FEEDFUN DISABLED LINE 2" : Bool;   // CG Feedfun Disabled Line 2
      "CG READY START LINE 2" : Bool;   // CG Ready Start Line 2
      "CG WAIT TO ESTABLISH LINE 2" : Bool;   // CG Wait To Establish Line 2
      "FEEDFUNC READY START LINE 2" : Bool;   // Feedfunc Ready Start Line 2
      "FEEDFUN RUNNING LINE 2" : Bool;   // Feedfun Running Line 2
      "FEEDFUN WAIT TO ZERO LINE 2" : Bool;   // Feedfun Wait To Zero Line 2
      "Mixer Fault" : Bool;   // Mixer Fault
      "Pressure Low Fault" : Bool;   // Pressure Low Fault
      "Gasflow Fault" : Bool;   // Gasflow Fault
      "Discflow Fault" : Bool;   // Discflow Fault
      "FEEDER PROFINET MODE ACTIVE" : Bool;   // Feeder Profinet Mode Active
      "FEEDER LINE 1 NOT READY FAULT" : Bool;   // Feeder Line 1 Not Ready Fault
      "FEEDER LINE 2 NOT READY FAULT" : Bool;   // Feeder Line 2 Not Ready Fault
      "FEEDER PROFINET MODE ACTIVE FAULT" : Bool;
      "Powder Line Clogged Line 1 Fault" : Bool;   // Powder Line Clogged Line 1 Fault
      "Powder Line Clogged Line 2 Fault" : Bool;   // Powder Line Clogged Line 2 Fault
      "Gas Flow Below Low Limit Line 1 Fault" : Bool;   // Gas Flow Below Low Limit Line 1 Fault
      "Gas Flow Below Low Limit Line 2 Fault" : Bool;   // Gas Flow Below Low Limit Line 2 Fault
      "Disk Speed Below Low Limit Line 1 Fault" : Bool;   // Disk Speed Below Low Limit Line 1 Fault
      "Disk Speed Below Low Limit Line 2 Fault" : Bool;   // Disk Speed Below Low Limit Line 2 Fault
      "Stirrer Speed Below Low Limit Line 1 Fault" : Bool;   // Stirrer Speed Below Low Limit Line 1 Fault
      "Stirrer Speed Below Low Limit Line 2 Fault" : Bool;   // Stirrer Speed Below Low Limit Line 2 Fault
      "Gas Flow Above High Limit Line 1 Fault" : Bool;   // Gas Flow Above High Limit Line 1 Fault
      "Gas Flow Above High Limit Line 2 Fault" : Bool;   // Gas Flow Above High Limit Line 2 Fault
      "Disk Speed Above High Limit Line 1 Fault" : Bool;   // Disk Speed Above High Limit Line 1 Fault
      "Disk Speed Above High Limit Line 2 Fault" : Bool;   // Disk Speed Above High Limit Line 2 Fault
      "Stirrer Speed Above High Limit Line 1 Fault" : Bool;   // Stirrer Speed Above High Limit Line 1 Fault
      "Stirrer Speed Above High Limit Line 2 Fault" : Bool;   // Stirrer Speed Above High Limit Line 2 Fault
      "Hopper Temperature Above High Limit Line 1 Fault" : Bool;   // Hopper Temperature Above High Limit Line 1 Fault
      "Hopper Temperature Above High Limit Line 2 Fault" : Bool;   // Hopper Temperature Above High Limit Line 2 Fault
      "Carrier Gas Inlet Pressure Too Low Line 1 Fault" : Bool;   // Carrier Gas Inlet Pressure Too Low Line 1 Fault
      "Carrier Gas Inlet Pressure Too Low Line 2 Fault" : Bool;   // Carrier Gas Inlet Pressure Too Low Line 2 Fault
      "Disk Motor Plugged In And Ready Line 1 Fault" : Bool;   // Disk Motor Plugged In And Ready Line 1 Fault
      "Disk Motor Plugged In And Ready Line 2 Fault" : Bool;   // Disk Motor Plugged In And Ready Line 2 Fault
      "Stirrer Plugged In And Ready Line 1 Fault" : Bool;   // Stirrer Plugged In And Ready Line 1 Fault
      "Stirrer Plugged In And Ready Line 2 Fault" : Bool;   // Stirrer Plugged In And Ready Line 2 Fault
      "Communication Running Line 1 Fault" : Bool;   // Communication Running Line 1 Fault
      "Communication Running Line 2 Fault" : Bool;   // Communication Running Line 2 Fault
      "Gas Flow Line 1 Under Warning" : Bool;   // Gas Flow Line 1 Under Warning
      "Gas Flow Line 2 Under Warning" : Bool;   // Gas Flow Line 2 Under Warning
      "Disk Speed Line 1 Under Warning" : Bool;   // Disk Speed Line 1 Under Warning
      "Disk Speed Line 2 Under Warning" : Bool;   // Disk Speed Line 2 Under Warning
      "Stirrer Speed Line 1 Under Warning" : Bool;   // Stirrer Speed Line 1 Under Warning
      "Stirrer Speed Line 2 Under Warning" : Bool;   // Stirrer Speed Line 2 Under Warning
      "Gas Flow Line 1 Over Warning" : Bool;   // Gas Flow Line 1 Over Warning
      "Gas Flow Line 2 Over Waning" : Bool;   // Gas Flow Line 2 Over Waning
      "Disk Speed Line 1 Over Warning" : Bool;   // Disk Speed Line 1 Over Warning
      "Disk Speed Line 2 Over Warning" : Bool;   // Disk Speed Line 2 Over Warning
      "Stirrer Speed Line 1 Over Warning" : Bool;   // Stirrer Speed Line 1 Over Warning
      "Stirrer Speed Line 2 Over Warning" : Bool;   // Stirrer Speed Line 2 Over Warning
      "Feeding Mode Gravimetric Line 1 Selected Warning" : Bool;   // Feeding Mode Gravimetric Line 1 Selected Warning
      "Feeding Mode Gravimetric Line 2 Selected Warning" : Bool;   // Feeding Mode Gravimetric Line 2 Selected Warning
      "CARRIER GAS IS RUNNING LINE 1" : Bool;   // Carrier Gas Is Running Line 1
      "CARRIER GAS IS OFFLINE 1" : Bool;   // Carrier Gas Is Off Line 1
      "CARRIER GAS IS RUNNING LINE 2" : Bool;   // Carrier Gas Is Running Line 2
      "CARRIER GAS IS OFFLINE 2" : Bool;   // Carrier Gas Is Off Line 2
      "Start General Conditions Help" : Bool;   // Start General Conditions Help
      "Start Initial Conditions Help" : Bool;   // Start Initial Conditions Help
      "Stop General Conditions Help" : Bool;   // Stop General Conditions Help
      "Stop Initial Conditions Help" : Bool;   // Stop Initial Conditions Help
      Fault : Bool;   // Fault
      "HMI Start" : Bool;   // HMI Start
      "HMI Stop" : Bool;   // HMI Stop
      "HMI Turned On" : Bool;   // HMI Turned On
      "HMI Turned Off" : Bool;   // HMI Turned Off
      "HMI Turning On" : Bool;   // HMI Turning On
      "HMI Turning Off" : Bool;   // HMI Turning Off
      "HMI Start Conditions" : Bool;   // HMI Start Conditions
      "HMI Stop Conditions" : Bool;   // HMI Stop Conditions
      "HMI Select G/Min Mode" : Bool;   // HMI Select G/Min Mode
      "HMI Turn On Powder Switch Nozzle" : Bool;   // HMI Turn On Powder Switch Nozzle
      "HMI Turn Off Powder Switch Nozzle" : Bool;   // HMI Turn Off Powder Switch Nozzle
      "HMI Switch On Profinet" : Bool;   // HMI Switch On Profinet
      "HMI Switch Off Profinet" : Bool;   // HMI Switch Off Profinet
      "HMI Set Temporal Disc RPMS" : Bool;   // HMI Set Temporal Disc RPMS
      "HMI Set Temporal Hopper Feedrate" : Bool;   // HMI Set Temporal Hopper Feedrate
      "HMI Set Temporal Gasflow" : Bool;   // HMI Set Temporal Gasflow
      "HMI Set Temporal Mixer" : Bool;   // HMI Set Temporal Mixer
      "HMI Actual Values Disc RPMS" : Bool;   // HMI Actual Values Disc RPMS
      "HMI Actual Values Hopper Feedrate" : Bool;   // HMI Actual Values Hopper Feedrate
      "HMI Actual Values Gasflow" : Bool;   // HMI Actual Values Gasflow
   END_STRUCT;
END_TYPE

TYPE "POWDER FEEDER HEATER JKT"
// stored: IsFailsafeCompliant false
   STRUCT
      START_GENERAL_CONDITIONS : Bool;   // Start General Conditions / START GENERAL CONDITIONS
      START_INITIAL_CONDITIONS_LINE_1 : Bool;   // Start Initial Conditions / START INITIAL CONDITIONS LINE 1
      START_INITIAL_CONDITIONS_LINE_2 : Bool;   // Start Initial Conditions / START INITIAL CONDITIONS LINE 2
      START_MANUAL_REQUEST_LINE_1 : Bool;   // Start Manual Request / START MANUAL REQUEST LINE 1
      START_MANUAL_REQUEST_LINE_2 : Bool;   // Start Manual Request / START MANUAL REQUEST LINE 2
      START_AUTO_REQUEST : Bool;   // Start Auto Request / START AUTO REQUEST
      START_GLOBAL_REQUEST_LINE_1 : Bool;   // Start Global Request / START GLOBAL REQUEST LINE 1
      START_GLOBAL_REQUEST_LINE_2 : Bool;   // Start Global Request / START GLOBAL REQUEST LINE 2
      START_COMMAND_LINE_1 : Bool;   // Start Command / START COMMAND LINE 1
      START_COMMAND_LINE_2 : Bool;   // Start Command / START COMMAND LINE 2
      START_LINE_1 : Bool;   // Start / START LINE 1
      START_LINE_2 : Bool;   // Start / START LINE 2
      FEEDBACK_ON_LINE_1 : Bool;   // Feedback On / FEEDBACK ON LINE 1
      FEEDBACK_ON_LINE_2 : Bool;   // Feedback On / FEEDBACK ON LINE 2
      STOP_GENERAL_CONDITIONS : Bool;   // Stop General Conditions / STOP GENERAL CONDITIONS
      STOP_INITIAL_CONDITIONS_LINE_1 : Bool;   // Stop Initial Conditions / STOP INITIAL CONDITIONS LINE 1
      STOP_INITIAL_CONDITIONS_LINE_2 : Bool;   // Stop Initial Conditions / STOP INITIAL CONDITIONS LINE 2
      STOP_MANUAL_REQUEST_LINE_1 : Bool;   // Stop Manual Request / STOP MANUAL REQUEST LINE 1
      STOP_MANUAL_REQUEST_LINE_2 : Bool;   // Stop Manual Request / STOP MANUAL REQUEST LINE 2
      STOP_AUTO_REQUEST : Bool;   // Stop Auto Request / STOP AUTO REQUEST
      STOP_GLOBAL_REQUEST_LINE_1 : Bool;   // Stop Global Request / STOP GLOBAL REQUEST LINE 1
      STOP_GLOBAL_REQUEST_LINE_2 : Bool;   // Stop Global Request / STOP GLOBAL REQUEST LINE 2
      STOP_COMMAND_LINE_1 : Bool;   // Stop Command / STOP COMMAND LINE 1
      STOP_COMMAND_LINE_2 : Bool;   // Stop Command / STOP COMMAND LINE 2
      STOP_LINE_1 : Bool;   // Stop / STOP LINE 1
      STOP_LINE_2 : Bool;   // Stop / STOP LINE 2
      FEEDBACK_OFF_LINE_1 : Bool;   // Feedback Off / FEEDBACK OFF LINE 1
      FEEDBACK_OFF_LINE_2 : Bool;   // Feedback Off / FEEDBACK OFF LINE 2
      START_GENERAL_CONDITIONS_HELP : Bool;   // Start General Conditions Help
      START_INITIAL_CONDITIONS_HELP : Bool;   // Start Initial Conditions Help
      STOP_GENERAL_CONDITIONS_HELP : Bool;   // Stop General Conditions Help
      STOP_INITIAL_CONDITIONS_HELP : Bool;   // Stop Initial Conditions Help
      FAULT : Bool;   // Fault
   END_STRUCT;
END_TYPE

